# B&R Automation Studio project VisionSample (part 2)

#### brdkSTR.fun
```iecst
FUNCTION brdkStrAppendUdintToA : DINT (*Appends an UDINT to the end of a string. $RETURN=length;Length of the string.*) (*$GROUP=User,$CAT=User,$GROUPICON=User.png,$CATICON=User.png*)
	VAR_INPUT
		value : UDINT; (*UDINT value to be converted.*)
		pString : UDINT; (*String pointer to source string.*)
		base : USINT; (*0,10 = decimal, 2 = binary, 16 = hex.*)
		position : DINT; (*Append position. Negative numbers will count from end of string.*)
	END_VAR
END_FUNCTION

FUNCTION brdkStrAToDint : DINT (*Converts a string to a DINT type. $RETURN=value;DINT value.*) (*$GROUP=User,$CAT=User,$GROUPICON=User.png,$CATICON=User.png*)
	VAR_INPUT
		pString : UDINT; (*String pointer to source string.*)
		base : USINT; (*0,10 = decimal, 2 = binary, 16 = hex.*)
	END_VAR
END_FUNCTION

FUNCTION brdkStrAToUdint : UDINT (*Converts a string to an UDINT type. $RETURN=value;UDINT value.*) (*$GROUP=User,$CAT=User,$GROUPICON=User.png,$CATICON=User.png*)
	VAR_INPUT
		pString : UDINT; (*String pointer to source string.*)
		base : USINT; (*0,10 = decimal, 2 = binary, 16 = hex.*)
	END_VAR
END_FUNCTION

FUNCTION brdkStrCat : UDINT (*Appends a copy of the source string to the end of the destination string. $RETURN=address;Address after the string.*) (*$GROUP=User,$CAT=User,$GROUPICON=User.png,$CATICON=User.png*)
	VAR_INPUT
		pDestination : UDINT; (*Destination string pointer.*)
		pSource : UDINT; (*Source string pointer.*)
	END_VAR
END_FUNCTION

FUNCTION brdkStrCatAtChar : DINT (*Appends a copy of the source string to the char position of the destination string. $RETURN=index;Index in destination string where the source string is appended. -1 if char is not found.*) (*$GROUP=User,$CAT=User,$GROUPICON=User.png,$CATICON=User.png*)
	VAR_INPUT
		pDestination : UDINT; (*Destination string pointer.*)
		pSource : UDINT; (*Source string pointer.*)
		pChar : UDINT; (*Char pointer.*)
		direction : DINT; (*0 = first appearance of char, -1 = last appearance of char.*)
		greedy : BOOL; (*If true the source string is appended to the char position. If false the char is still present in the destination string.*)
	END_VAR
END_FUNCTION

FUNCTION brdkStrCharAt : USINT (*Returns the character at the specified index. $RETURN=coding;ASCII coding of the char.*) (*$GROUP=User,$CAT=User,$GROUPICON=User.png,$CATICON=User.png*)
	VAR_INPUT
		pString : UDINT; (*String pointer to source string.*)
		index : UDINT; (*Look up index.*)
		pChar : UDINT; (*Char pointer to char to look up.*)
	END_VAR
END_FUNCTION

FUNCTION brdkStrCharCount : DINT (*Finds how many times a character appears in a string. $RETURN=count;Char count. -1 if error.*) (*$GROUP=User,$CAT=User,$GROUPICON=User.png,$CATICON=User.png*)
	VAR_INPUT
		pString : UDINT; (*String pointer to source string.*)
		pChar : UDINT; (*Pointer to search char.*)
	END_VAR
END_FUNCTION

FUNCTION brdkStrCmp : DINT (*Compares character(s) from string1 to string2. $RETURN=result;0 means that the two string are equal.*)
	VAR_INPUT
		pString1 : UDINT; (*String1 pointer.*)
		pString2 : UDINT; (*String2 pointer.*)
	END_VAR
END_FUNCTION

FUNCTION brdkStrCpy : UDINT (*Copies a string to another string. $RETURN=address;Address after the string.*) (*$GROUP=User,$CAT=User,$GROUPICON=User.png,$CATICON=User.png*)
	VAR_INPUT
		pDestination : UDINT; (*Destination string pointer.*)
		pSource : UDINT; (*Source string pointer.*)
	END_VAR
END_FUNCTION

FUNCTION brdkStrCrc32 : UDINT (*Calculates a CRC32 checksum based on the input string. $RETURN=checksum;Checksum of the string.*) (*$GROUP=User,$CAT=User,$GROUPICON=User.png,$CATICON=User.png*)
	VAR_INPUT
		pString : UDINT; (*String pointer.*)
	END_VAR
END_FUNCTION

FUNCTION brdkStrDintToA : DINT (*Converts a DINT into a STRING type. $RETURN=length;Length of the string.*) (*$GROUP=User,$CAT=User,$GROUPICON=User.png,$CATICON=User.png*)
	VAR_INPUT
		value : DINT; (*DINT value to be converted.*)
		pString : UDINT; (*String pointer to source string.*)
		base : USINT; (*0,10 = decimal, 2 = binary, 16 = hex.*)
	END_VAR
END_FUNCTION

FUNCTION brdkStrEncode : DINT (*Encodes a string into different formats. $RETURN=address;Address after the string.*) (*$GROUP=User,$CAT=User,$GROUPICON=User.png,$CATICON=User.png*)
	VAR_INPUT
		pDestination : UDINT; (*Destination string pointer.*)
		pSource : UDINT; (*Source string pointer.*)
		format : USINT; (*0 = UTF-8*)
	END_VAR
END_FUNCTION

FUNCTION brdkStrFill : DINT (*Inserts amount of character(s) to the specified position of the string. $RETURN=length;Length of the string. -1 if error.*) (*$GROUP=User,$CAT=User,$GROUPICON=User.png,$CATICON=User.png*)
	VAR_INPUT
		pString : UDINT; (*String pointer to source string.*)
		amount : DINT; (*Fill char amount.*)
		pChar : UDINT; (*Fill char. If 0 whitespace is used.*)
		position : DINT; (*Fill position. Negative numbers will count from end of string.*)
	END_VAR
END_FUNCTION

FUNCTION brdkStrFillUp : DINT (*Fills x amount of character(s) to the specified position of the string. $RETURN=amount;Amount of chars filled. -1 if error.*) (*$GROUP=User,$CAT=User,$GROUPICON=User.png,$CATICON=User.png*)
	VAR_INPUT
		pString : UDINT; (*String pointer to source string.*)
		maxLength : DINT; (*Maximum length of the string.*)
		pChar : UDINT; (*Fill char. If 0 whitespace is used.*)
		position : DINT; (*Fill position. Negative numbers will count from end of string.*)
	END_VAR
END_FUNCTION

FUNCTION brdkStrIndexOf : DINT (*Returns the index within this string of the first or last occurrence of the specified character. $RETURN=index;Index of the char. -1 if char is not found.*) (*$GROUP=User,$CAT=User,$GROUPICON=User.png,$CATICON=User.png*)
	VAR_INPUT
		pString : UDINT; (*String pointer to source string.*)
		pChar : UDINT; (*Char pointer to char to look up.*)
		direction : DINT; (*0 = search from left, -1 = search from right.*)
	END_VAR
END_FUNCTION

FUNCTION brdkStrInsertAtPos : DINT (*Inserts a string into another string at a specified position. $RETURN=length;Length of the string. -1 if error.*) (*$GROUP=User,$CAT=User,$GROUPICON=User.png,$CATICON=User.png*)
	VAR_INPUT
		pString : UDINT; (*String pointer to source string.*)
		pInsert : UDINT; (*String pointer to insert string.*)
		position : DINT; (*Insert position. Negative numbers will count from end of string.*)
	END_VAR
END_FUNCTION

FUNCTION brdkStrIsAlphabet : BOOL (*Returns false or true depending of all characters are present in the alphabet. $RETURN=false/true; a..z = true.*) (*$GROUP=User,$CAT=User,$GROUPICON=User.png,$CATICON=User.png*)
	VAR_INPUT
		pString : UDINT; (*String pointer.*)
	END_VAR
END_FUNCTION

FUNCTION brdkStrIsDigit : BOOL (*Returns false or true depending of all characters are digits. $RETURN=false/true; 0..9 = true.*) (*$GROUP=User,$CAT=User,$GROUPICON=User.png,$CATICON=User.png*)
	VAR_INPUT
		pString : UDINT; (*String pointer.*)
	END_VAR
END_FUNCTION

FUNCTION brdkStrIsEmpty : BOOL (*Returns false or true depending of characters are present in the first position of the string. $RETURN=false/true;Position [0] = /0 = false. Position [0] != /0 = true.*) (*$GROUP=User,$CAT=User,$GROUPICON=User.png,$CATICON=User.png*)
	VAR_INPUT
		pString : UDINT; (*String pointer.*)
	END_VAR
END_FUNCTION

FUNCTION brdkStrJoin : DINT (*Joins elements from a string array into a string with a delimiter. $RETURN=length;Length of the string or error codes.*) (*$GROUP=User,$CAT=User,$GROUPICON=User.png,$CATICON=User.png*)
	VAR_INPUT
		pString : UDINT; (*String pointer to destination string.*)
		pArray : UDINT; (*Pointer to source string array.*)
		pDelimiter : UDINT; (*Delimiter char. If 0 whitespace is used. The delimiter can only be 1 char long.*)
		sizeOfArray : UDINT; (*Max. size of the string array. Size means number of elements in array.*)
		sizeOfArrayString : UDINT; (*Max. size of strings in the array.*)
		sizeOfString : UDINT; (*Max. size of destination string.*)
	END_VAR
END_FUNCTION

FUNCTION brdkStrLen : DINT (*Returns the number of characters in a string. Stops at \0. $RETURN=length;length of the string*) (*$GROUP=User,$CAT=User,$GROUPICON=User.png,$CATICON=User.png*)
	VAR_INPUT
		pString : UDINT; (*String pointer.*)
	END_VAR
END_FUNCTION

FUNCTION brdkStrMemClear : UDINT (*Fills amount of 0 to destination. $RETURN=address;Address after the destination.*) (*$GROUP=User,$CAT=User,$GROUPICON=User.png,$CATICON=User.png*)
	VAR_INPUT
		pDestination : UDINT; (*Destination pointer.*)
		amount : UDINT; (*Amount of character(s) to be initialized.*)
	END_VAR
END_FUNCTION

FUNCTION brdkStrMemCmp : DINT (*Compares amount of character(s) from area1 to area2. $RETURN=result;0 means that the two areas are equal.*) (*$GROUP=User,$CAT=User,$GROUPICON=User.png,$CATICON=User.png*)
	VAR_INPUT
		pArea1 : UDINT; (*Area1 pointer.*)
		pArea2 : UDINT; (*Area2 pointer.*)
		amount : UDINT; (*Amount of character(s) to be comared.*)
	END_VAR
END_FUNCTION

FUNCTION brdkStrMemCpy : UDINT (*Copies amount of character(s) from source to destination. $RETURN=address;Address after the destination.*) (*$GROUP=User,$CAT=User,$GROUPICON=User.png,$CATICON=User.png*)
	VAR_INPUT
		pDestination : UDINT; (*Destination pointer.*)
		pSource : UDINT; (*Source pointer.*)
		amount : UDINT; (*Amount of character(s) to be copied.*)
	END_VAR
END_FUNCTION

FUNCTION brdkStrMemMove : UDINT (*Moves amount of character(s) from source to destination. $RETURN=address;Address after the destination.*) (*$GROUP=User,$CAT=User,$GROUPICON=User.png,$CATICON=User.png*)
	VAR_INPUT
		pDestination : UDINT; (*Destination pointer.*)
		pSource : UDINT; (*Source pointer.*)
		amount : UDINT; (*Amount of character(s) to be moved.*)
	END_VAR
END_FUNCTION

FUNCTION brdkStrMemSet : UDINT (*Fills amount of character(s) to destination. $RETURN=address;Address after the destination.*) (*$GROUP=User,$CAT=User,$GROUPICON=User.png,$CATICON=User.png*)
	VAR_INPUT
		pDestination : UDINT; (*Destination pointer.*)
		value : USINT; (*Initialization value.*)
		amount : UDINT; (*Amount of character(s) to be initialized.*)
	END_VAR
END_FUNCTION

FUNCTION brdkStrMove : UDINT (*Moves a string to another string. $RETURN=address;Address after the string.*) (*$GROUP=User,$CAT=User,$GROUPICON=User.png,$CATICON=User.png*)
	VAR_INPUT
		pDestination : UDINT; (*Destination string pointer.*)
		pSource : UDINT; (*Source string pointer.*)
	END_VAR
END_FUNCTION

FUNCTION brdkStrNCpy : UDINT (*Copies a string to another string. If the function encounters a null character in the source string, the function will add null characters to the destination string until amount character(s) have been written. $RETURN=address;Address after the string.*) (*$GROUP=User,$CAT=User,$GROUPICON=User.png,$CATICON=User.png*)
	VAR_INPUT
		pDestination : UDINT; (*Destination string pointer.*)
		pSource : UDINT; (*Source string pointer.*)
		amount : UDINT; (*Amount of character(s) to be moved.*)
	END_VAR
END_FUNCTION

FUNCTION brdkStrRemove : UDINT (*Removes character(s) from a string from a specified position. $RETURN=address;Address after the string.*) (*$GROUP=User,$CAT=User,$GROUPICON=User.png,$CATICON=User.png*)
	VAR_INPUT
		pString : UDINT; (*Source string pointer.*)
		start : DINT; (*Index of where to start in the string. Negative numbers start from the end of the string.*)
		length : DINT; (*0 means to the end of the string. Negative length is subtracted from the end of the string. Is start is negative length is subtracted from the start of the string. *)
	END_VAR
END_FUNCTION

FUNCTION brdkStrRepeat : DINT (*Repeats a string a specified number of times. $RETURN=length;Length of the string.*) (*$GROUP=User,$CAT=User,$GROUPICON=User.png,$CATICON=User.png*)
	VAR_INPUT
		pString : UDINT; (*String pointer to source string.*)
		times : DINT; (*Number of times the string should be repeated.*)
	END_VAR
END_FUNCTION

FUNCTION brdkStrReplace : DINT (*Replaces some characters with some other characters in a string. $RETURN=number;Number of replacements done.*) (*$GROUP=User,$CAT=User,$GROUPICON=User.png,$CATICON=User.png*)
	VAR_INPUT
		pString : UDINT; (*String pointer to source string.*)
		pFind : UDINT; (*String pointer to find string.*)
		pReplace : UDINT; (*String pointer to replacement string:*)
	END_VAR
END_FUNCTION

FUNCTION brdkStrReverse : DINT (*Reverses a string from start position to end position. $RETURN=count;Number of reverses done. -1 if error.*) (*$GROUP=User,$CAT=User,$GROUPICON=User.png,$CATICON=User.png*)
	VAR_INPUT
		pString : UDINT; (*String pointer to source string.*)
		startPosition : DINT; (*Start position. Must be a positive number and less than length.*)
		endPosition : DINT; (*End position. Must be less than length unless it's a negative numbers which will count from end of string.*)
	END_VAR
END_FUNCTION

FUNCTION brdkStrReverseWords : DINT (*Reverses words in a string. $RETURN=count;Number of words reversed.*) (*$GROUP=User,$CAT=User,$GROUPICON=User.png,$CATICON=User.png*)
	VAR_INPUT
		pString : UDINT; (*String pointer to source string.*)
	END_VAR
END_FUNCTION

FUNCTION brdkStrSearch : DINT (*Searches a string for a specified string. $RETURN=position; Position of the match. -1 if no match.*) (*$GROUP=User,$CAT=User,$GROUPICON=User.png,$CATICON=User.png*)
	VAR_INPUT
		pString : UDINT; (*String pointer to source string.*)
		pSearchString : UDINT; (*String pointer to search string.*)
	END_VAR
END_FUNCTION

FUNCTION brdkStrSlice : DINT (*Slices a part of a string. $RETURN=length;Length of the string. -1 if error.*) (*$GROUP=User,$CAT=User,$GROUPICON=User.png,$CATICON=User.png*)
	VAR_INPUT
		pString : UDINT; (*String pointer to source string.*)
		start : DINT; (*Start position.*)
		end : DINT; (*End position.*)
	END_VAR
END_FUNCTION

FUNCTION brdkStrSplit : DINT (*Splits a string into an array of string using a seperator. $RETURN=count;Number of elements splitted or an error code.*) (*$GROUP=User,$CAT=User,$GROUPICON=User.png,$CATICON=User.png*)
	VAR_INPUT
		pArray : UDINT; (*Pointer to destination string array.*)
		pString : UDINT; (*String pointer to source string.*)
		pDelimiter : UDINT; (*Delimiter char. If 0 whitespace is used. The delimiter can only be 1 char long.*)
		sizeOfArray : UDINT; (*Max. size of the string array. Size means number of elements in array.*)
		sizeofArrayString : UDINT; (*Max. size of strings in the array.*)
		greedy : BOOL; (*Remove or keep the seperator from the string.*)
	END_VAR
END_FUNCTION

FUNCTION brdkStrSubDintSearch : DINT (*Returns a DINT based on a search. $RETURN=length;Length of the destination string. -1 if error.*) (*$GROUP=User,$CAT=User,$GROUPICON=User.png,$CATICON=User.png*)
	VAR_INPUT
		pSource : UDINT; (*Source string pointer.*)
		pStart : UDINT; (*String pointer for start search string.*)
		pEnd : UDINT; (*String pointer for end search string. The function will only search after the start string.*)
		startOffset : DINT; (*Offset for the start poition. If greedy = true offset is after the start has been removed.*)
		base : USINT; (*0,10 = decimal, 2 = binary, 16 = hex.*)
	END_VAR
END_FUNCTION

FUNCTION brdkStrSubStr : DINT (*Returns a part of a string. $RETURN=length;Length of the destination string. -1 if error.*) (*$GROUP=User,$CAT=User,$GROUPICON=User.png,$CATICON=User.png*)
	VAR_INPUT
		pDestination : UDINT; (*Destination string pointer.*)
		pSource : UDINT; (*Source string pointer.*)
		start : DINT; (*Index of where to start in the string. Negative numbers start from the end of the string.*)
		length : DINT; (*0 means to the end of the string. Negative length is subtracted from the end of the string. Is start is negative length is subtracted from the start of the string. *)
	END_VAR
END_FUNCTION

FUNCTION brdkStrSubStrSearch : BOOL (*Returns a part of a string based on a search. $RETURN=success;TRUE = success *) (*$GROUP=User,$CAT=User,$GROUPICON=User.png,$CATICON=User.png*)
	VAR_INPUT
		pDestination : UDINT; (*Destination string pointer.*)
		pSource : UDINT; (*Source string pointer.*)
		pStart : UDINT; (*String pointer for start search string.*)
		pEnd : UDINT; (*String pointer for end search string. The function will only search after the start string.*)
		startOffset : DINT; (*Offset for the start poition. If greedy = true offset is after the start has been removed.*)
		greedy : BOOL; (*Will add or remove the search strings from the destination string.*)
	END_VAR
END_FUNCTION

FUNCTION brdkStrToDec : DINT (*Converts a string of hexadecimal values to ASCII characters. $RETURN=length;Length of the string. -1 if error.*) (*$GROUP=User,$CAT=User,$GROUPICON=User.png,$CATICON=User.png*)
	VAR_INPUT
		pString : UDINT; (*String pointer to source string.*)
	END_VAR
END_FUNCTION

FUNCTION brdkStrToHex : DINT (*Converts a string of ASCII characters to hexadecimal values. $RETURN=length;Length of the string.*) (*$GROUP=User,$CAT=User,$GROUPICON=User.png,$CATICON=User.png*)
	VAR_INPUT
		pString : UDINT; (*String pointer to source string.*)
	END_VAR
END_FUNCTION

FUNCTION brdkStrToLowerCase : DINT (*Converts a string to lowercase letters. $RETURN=number;Number of characters changed.*) (*$GROUP=User,$CAT=User,$GROUPICON=User.png,$CATICON=User.png*)
	VAR_INPUT
		pString : UDINT; (*String pointer to source string.*)
	END_VAR
END_FUNCTION

FUNCTION brdkStrToUpperCase : DINT (*Converts a string to uppercase letters. $RETURN=number;Number of characters changed.*) (*$GROUP=User,$CAT=User,$GROUPICON=User.png,$CATICON=User.png*)
	VAR_INPUT
		pString : UDINT; (*String pointer to source string.*)
	END_VAR
END_FUNCTION

FUNCTION brdkStrToUpperCaseWords : DINT (*Convert the first character of each word to uppercase. (title()). $RETURN=number;Number of characters changed.*) (*$GROUP=User,$CAT=User,$GROUPICON=User.png,$CATICON=User.png*)
	VAR_INPUT
		pString : UDINT; (*String pointer to source string.*)
	END_VAR
END_FUNCTION

FUNCTION brdkStrTrim : DINT (*Removes whitespaces from a string. $RETURN=number;Number of whitespaces removed from string.*) (*$GROUP=User,$CAT=User,$GROUPICON=User.png,$CATICON=User.png*)
	VAR_INPUT
		pString : UDINT; (*String pointer to source string.*)
		direction : DINT; (*0 = both sides, 1 = left side only, -1 = right side only.*)
	END_VAR
END_FUNCTION

FUNCTION brdkStrUdintToA : DINT (*Converts an UDINT into a STRING type. $RETURN=length;Length of the string.*) (*$GROUP=User,$CAT=User,$GROUPICON=User.png,$CATICON=User.png*)
	VAR_INPUT
		value : UDINT; (*UDINT value to be converted.*)
		pString : UDINT; (*String pointer to source string.*)
		base : USINT; (*0,10 = decimal, 2 = binary, 16 = hex.*)
	END_VAR
END_FUNCTION

FUNCTION brdkStrWord : DINT (*Returns a word in a string given by a number and a delimiter. $RETURN=length;Length of the string.*) (*$GROUP=User,$CAT=User,$GROUPICON=User.png,$CATICON=User.png*)
	VAR_INPUT
		pDestination : UDINT; (*Destination string pointer.*)
		pSource : UDINT; (*Source string pointer.*)
		pDelimiter : UDINT; (*Delimiter char. If 0 whitespace is used. The delimiter can only be 1 char long.*)
		number : DINT; (*Word number in string. 1 = first word. -1 = last word.*)
		sizeOfString : UDINT; (*Max. size of destination string.*)
	END_VAR
END_FUNCTION
```

#### brdkStrAppendUdintToA.c
```c
#include <brdkSTR_func.h>

signed long brdkStrAppendUdintToA(unsigned long value, unsigned long pString, unsigned char base, signed long position) {
	signed long i,cnt=0,len = brdkStrLen(pString);
	signed long start = position > -1 ? position :len+position+1;
	unsigned char tmp;
	i=start;
	tmp = 0x30;
	base = !base ? 10 : base;	/* make sure base is not 0 */
	if (value != 0) {
		while (value > 0) {
			unsigned long rem = value % base;
			unsigned char tmp = (rem > 9)? (rem-10) + 0x41 : rem + 0x30;	/* 0x41 = A, 0x30 = 0*/
			brdkStrFill(pString,1,(unsigned long)&tmp,i++);
	       	value = value/base;
			cnt++;
		}
		brdkStrReverse(pString,start,--i);
		return len+cnt;
	}
	else {
		brdkStrFill(pString,1,(unsigned long)&tmp,i);
		return len+1;
	}
}
```

#### brdkStrAToDint.c
```c
#include <brdkSTR_func.h>

signed long brdkStrAToDint(unsigned long pString, unsigned char base) {
	/* check if string starts with a minus sign */
	if(((char*)pString)[0] == 0x2d) return -brdkStrAToUdint(pString+1,BRDK_STR_CONVERT_DECIMAL);
	else return brdkStrAToUdint(pString,base);
}
```

#### brdkStrAToUdint.c
```c
#include <brdkSTR_func.h>

unsigned long brdkStrAToUdint(unsigned long pString, unsigned char base) {
	signed long len = brdkStrLen(pString);
	return aToUdint(pString, len, base);
}
```

#### brdkStrCat.c
```c
#include <brdkSTR_func.h>

unsigned long brdkStrCat(unsigned long pDestination, unsigned long pSource) {
	unsigned long i=0,len = brdkStrLen(pSource), start = brdkStrLen(pDestination);
	for(i=0; i< len; i++) ((char*)pDestination)[start+i] = ((char*)pSource)[i];
	((char*)pDestination)[start+i] = 0;
	return pDestination+start+i;
}
```

#### brdkStrCatAtChar.c
```c
#include <brdkSTR_func.h>

signed long brdkStrCatAtChar(unsigned long pDestination, unsigned long pSource, unsigned long pChar, signed long direction, unsigned char greedy) {
	unsigned long i=0,len = brdkStrLen(pSource);
	signed long start = brdkStrIndexOf(pDestination,pChar,direction);
	if(start > -1) {
		start += !greedy;
		for(i=0; i< len; i++) ((char*)pDestination)[start+i] = ((char*)pSource)[i];
		((char*)pDestination)[start+i] = 0;
	}
	return start;
}
```

#### brdkStrCharAt.c
```c
#include <brdkSTR_func.h>

unsigned char brdkStrCharAt(unsigned long pString, unsigned long index, unsigned long pChar) {
	if(index < brdkStrLen(pString)) {
		*(char*)pChar = ((char*)pString)[index];
		return ((char*)pString)[index];
	}
	else {
		*(char*)pChar = 0;
		return 0;
	}
}
```

#### brdkStrCharCount.c
```c
#include <brdkSTR_func.h>

signed long brdkStrCharCount(unsigned long pString, unsigned long pChar) {
	signed long i=0, cnt=0;
	if(pChar != 0 && *(char*)pChar != 0) {
		while(((char*)pString)[i]) if(((char*)pString)[i++] == *(char*)pChar) cnt++;
	}
	else cnt = -1;
	return cnt;
}
```

#### brdkStrCmp.c
```c
#include <brdkSTR_func.h>

signed long brdkStrCmp(unsigned long pString1, unsigned long pString2) {
	unsigned long i=0;
	do if(((char*)pString1)[i] != ((char*)pString2)[i]) break;
	while(((char*)pString1)[i] != 0 && ((char*)pString2)[i++] != 0);
	return ((char*)pString1)[i]-((char*)pString2)[i];
}
```

#### brdkStrCpy.c
```c
#include <brdkSTR_func.h>

unsigned long brdkStrCpy(unsigned long pDestination, unsigned long pSource) {
	unsigned long i=0;
	do ((char*)pDestination)[i] = ((char*)pSource)[i];
	while(((char*)pSource)[i++] != 0);
	return pDestination+i;
}
```

#### brdkStrCrc32.c
```c
#include <brdkSTR_func.h>

unsigned long brdkStrCrc32(unsigned long pString) {
	int i=0, crc = 0xFFFFFFFF;
	unsigned int byte, c;
	const unsigned int g0 = 0xEDB88320, g1 = g0>>1,g2 = g0>>2, g3 = g0>>3, g4 = g0>>4, g5 = g0>>5, g6 = (g0>>6)^g0, g7 = ((g0>>6)^g0)>>1;
	while ((byte = ((char*)pString)[i]) != 0) {    /* Get next byte. */
		crc = crc ^ byte;
		c = ((crc<<31>>31) & g7) ^ ((crc<<30>>31) & g6) ^
			((crc<<29>>31) & g5) ^ ((crc<<28>>31) & g4) ^
			((crc<<27>>31) & g3) ^ ((crc<<26>>31) & g2) ^
			((crc<<25>>31) & g1) ^ ((crc<<24>>31) & g0);
		crc = ((unsigned)crc >> 8) ^ c;
		i++;
   }
   return ~crc;
}
```

#### brdkStrDintToA.c
```c
#include <brdkSTR_func.h>

signed long brdkStrDintToA(signed long value, unsigned long pString, unsigned char base) {
	if(value < 0) {
		((char*)pString)[0] = 0x2d; /* - sign */
		return brdkStrUdintToA(-value,pString+1,BRDK_STR_CONVERT_DECIMAL)+1;
	}
	else return brdkStrUdintToA(value,pString,base);
}
```

#### brdkStrEncode.c
```c
#include <brdkSTR_func.h>

signed long brdkStrEncode(unsigned long pDestination, unsigned long pSource, unsigned char format) {
	unsigned long i=0;
	switch(format) {
		case BRDK_STR_UTF_8:

			do ((unsigned char*)pDestination)[i] = ((unsigned char*)pSource)[i] <= 127 ? ((unsigned char*)pSource)[i] : ((unsigned char*)pSource)[i] + 35;
			while(((char*)pSource)[i++] != 0);
			return pDestination+i;
			break;

		default:
			return -1;
			break;
	}
}
```

#### brdkStrFill.c
```c
#include <brdkSTR_func.h>

signed long brdkStrFill(unsigned long pString, signed long amount, unsigned long pChar, signed long position) {
	signed long i,j, len = brdkStrLen(pString), tmpPos;
	char ch;
	i = len+amount;
	j = len;
	ch = pChar != 0 && *(char*)pChar != 0 ? *(char*)pChar : 0x20;	/* white space is default */
	tmpPos = position >= 0 ? position : len + 1 + position;
	if(tmpPos > -1) {
		while(j>=tmpPos) ((char*)pString)[i--] = ((char*)pString)[j--];
		while(i>=tmpPos) ((char*)pString)[i--] = ch;
		return len+amount;
	}
	else return -1;
}
```

#### brdkStrFillUp.c
```c
#include <brdkSTR_func.h>

signed long brdkStrFillUp(unsigned long pString, signed long maxLength, unsigned long pChar, signed long position) {
	signed long amount = maxLength-brdkStrLen(pString);
	if(amount > 0) {
		if(brdkStrFill(pString, amount, pChar, position) != -1) return amount;
		else return -1;
	}
	return 0;
}
```

#### brdkStrIndexOf.c
```c
#include <brdkSTR_func.h>

signed long brdkStrIndexOf(unsigned long pString, unsigned long pChar, signed long direction) {
	signed long i;
	if(direction > -1) {
		i = 0;
		while(((char*)pString)[i]) {
			if(((char*)pString)[i] == ((char*)pChar)[0]) break;
			else i++;
		}
		if(((char*)pString)[i] != 0) return i;
		else return -1;
	}
	else {
		i = brdkStrLen(pString)-1;
		while(((char*)pString)[i] && i > -1) if(((char*)pString)[i--] == ((char*)pChar)[0]) break;
		if(((char*)pString)[i] != 0) return ++i;
		else return -1;
	}
}
```

#### brdkStrInsertAtPos.c
```c
#include <brdkSTR_func.h>

signed long brdkStrInsertAtPos(unsigned long pString, unsigned long pInsert, signed long position) {
	signed long i,j, len = brdkStrLen(pString), lenIns = brdkStrLen(pInsert), tmpPos;
	if(lenIns > 0) {
		if(len==0 && (position==0 || position==-1)){
			i=0;
			while(((char*)pInsert)[i]) {
				((char*)pString)[i] = ((char*)pInsert)[i];
				i++;
			}
			((char*)pString)[i] = 0;
			len = i;
		}
		else if(position <= len) {
			i = len+lenIns;
			j = len;
			tmpPos = position >= 0 ? position : len + 1 + position;
			if(tmpPos > -1) {
				while(j>=tmpPos) ((char*)pString)[i--] = ((char*)pString)[j--];
				j=lenIns-1;
				while(i>=tmpPos) ((char*)pString)[i--] = ((char*)pInsert)[j--];
				len+=lenIns;
			}
			else len = -1;
		}
	}
	return len;
}
```

#### brdkStrIsAlphabet.c
```c
#include <brdkSTR_func.h>

unsigned char brdkStrIsAlphabet(unsigned long pString) {
	unsigned long len = 0;
	while(((char*)pString)[len]) {
		if (((char*)pString)[len] > 0x5A) {	/* is it larger that Z */
			if(((char*)pString)[len] < 0x61 || 0x7a < ((char*)pString)[len]) return 0;
		}
		else if(((char*)pString)[len] < 0x41) return 0;		/* is it smaller than A */
		len++;
	}
	return 1;
}
```

#### brdkStrIsDigit.c
```c
#include <brdkSTR_func.h>

unsigned char brdkStrIsDigit(unsigned long pString) {
	unsigned long len = 0;
	while(((char*)pString)[len]) {
		if (((char*)pString)[len] < 0x30 || 0x39 < ((char*)pString)[len]) return 0;
		len++;
	}
	return 1;
}
```

#### brdkStrIsEmpty.c
```c
#include <brdkSTR_func.h>

unsigned char brdkStrIsEmpty(unsigned long pString) {
	return ((char*)pString)[0] == 0;
}
```

#### brdkStrJoin.c
```c
#include <brdkSTR_func.h>

signed long brdkStrJoin(unsigned long pString, unsigned long pArray, unsigned long pDelimiter, unsigned long sizeOfArray, unsigned long sizeOfArrayString, unsigned long sizeOfString) {
	unsigned long sIdx = 0, pArr = pArray, aIdx = 0;
	if(pArray != 0 && pString != 0 && sizeOfArray != 0 && sizeOfArrayString != 0) {		/* check all pointers are set */
		if(pDelimiter == 0) pDelimiter = (unsigned long)" ";							/* use white space is delimiter pointer is 0 */
		while(((char*)pArr)[0] != 0) {													/* continue until we find the first empty array string */
			if(((char*)pArr)[aIdx] != 0) {
				((char*)pString)[sIdx++] = ((char*)pArr)[aIdx++];						/* copy string data */
				if(sIdx >= sizeOfString) return -2;										/* destination string too small */
			}
			else {
				pArr += sizeOfArrayString;												/* jump to the next array element */
				aIdx = 0;
				((char*)pString)[sIdx++] = ((char*)pDelimiter)[0];						/* insert delimiter */
				if(sIdx >= sizeOfString) return -2;										/* destination string too small */
				if(pArr > (pArray + sizeOfArray)) {										/* we hit the end of the array */
					break;
				}
			}
		}
		if(sIdx == 0) return 0;															/* nothing copied */
		sIdx--;
		((char*)pString)[sIdx] = 0;														/* end the string. -e because we inserted a delimiter at the end */
		return sIdx;
	}
	else return -1;
	return -4;
}
```

#### brdkStrLen.c
```c
#include <brdkSTR_func.h>

signed long brdkStrLen(unsigned long pString) {
	unsigned long len = 0;
	while(((char*)pString)[len]) len++;	/* makes a little strlen */
	return len;
}
```

#### brdkStrMemClear.c
```c
#include <brdkSTR_func.h>

unsigned long brdkStrMemClear(unsigned long pDestination, unsigned long amount) {
	return brdkStrMemSet(pDestination,0,amount);
}
```

#### brdkStrMemCmp.c
```c
#include <brdkSTR_func.h>

signed long brdkStrMemCmp(unsigned long pString1, unsigned long pString2, unsigned long amount) {
	unsigned long i=0;
	for(i=0; i< amount; i++) if(((char*)pString1)[i] != ((char*)pString2)[i]) break;
	return ((char*)pString1)[i]-((char*)pString2)[i];
}
```

#### brdkStrMemCpy.c
```c
#include <brdkSTR_func.h>

unsigned long brdkStrMemCpy(unsigned long pDestination, unsigned long pSource, unsigned long amount) {
	unsigned long i=0;
	for(i=0; i< amount; i++) ((char*)pDestination)[i] = ((char*)pSource)[i];
	return pDestination+amount;
}
```

#### brdkStrMemMove.c
```c
#include <brdkSTR_func.h>

unsigned long brdkStrMemMove(unsigned long pDestination, unsigned long pSource, unsigned long amount) {
	unsigned long i=0;
	char buffer[amount];	/* if the destination and source is the same string we need a buffer */
	for(i=0; i< amount; i++) buffer[i] = ((char*)pSource)[i];
	for(i=0; i< amount; i++) ((char*)pDestination)[i] = buffer[i];
	return pDestination+amount;
}
```

#### brdkStrMemSet.c
```c
#include <brdkSTR_func.h>

unsigned long brdkStrMemSet(unsigned long pDestination, unsigned char value, unsigned long amount) {
	unsigned long i=0;
	for(i=0; i< amount; i++) ((char*)pDestination)[i] = value;
	return pDestination+amount;
}
```

#### brdkStrMove.c
```c
#include <brdkSTR_func.h>

unsigned long brdkStrMove(unsigned long pDestination, unsigned long pSource) {
	return brdkStrMemMove(pDestination,pSource,brdkStrLen(pSource));
}
```

#### brdkStrNCpy.c
```c
#include <brdkSTR_func.h>

unsigned long brdkStrNCpy(unsigned long pDestination, unsigned long pSource, unsigned long amount) {
	unsigned long i=0;
	for(i=0; i< amount; i++) {
		if(((char*)pSource)[i]) ((char*)pDestination)[i] = ((char*)pSource)[i];
		else ((char*)pDestination)[i] = 0;
	}
	return pDestination+amount;
}
```

#### brdkStrRemove.c
```c
#include <brdkSTR_func.h>

unsigned long brdkStrRemove(unsigned long pString, signed long start, signed long length) {
	signed long end, len=0;
	if(start < 0) {
		len = brdkStrLen(pString);
		if(length<1) {
			len = start;
			start = length*(-1);
			length = brdkStrLen(pString)-start+len+1;
		}
		else start = len+start-length+1;
	}
	else if(length<1) length = brdkStrLen(pString)-start+length;
	end = start+length;
	while(((char*)pString)[end]) ((char*)pString)[start++] = ((char*)pString)[end++];
	((char*)pString)[start] = 0;
	return pString+start+1;
}
```

#### brdkStrRepeat.c
```c
#include <brdkSTR_func.h>

signed long brdkStrRepeat(unsigned long pString, signed long times) {
	signed long i,j,t,len = brdkStrLen(pString);
	j=len;
	for(t=0; t < times; t++) {
		for(i=0; i< len; i++) ((char*)pString)[j+i] = ((char*)pString)[i];
		j += len;
	}
	((char*)pString)[j] = 0;
	return j;
}
```

#### brdkStrReplace.c
```c
#include <brdkSTR_func.h>

signed long brdkStrReplace(unsigned long pString, unsigned long pFind, unsigned long pReplace) {
	signed long i=0, cnt=0, lenF = brdkStrLen(pFind), lenR = brdkStrLen(pReplace);
	i = brdkStrSearch(pString,pFind);
	while(i > -1) {
		brdkStrRemove(pString,i,lenF);
		brdkStrInsertAtPos(pString,pReplace,i);
		pString += i + lenR;
		i = brdkStrSearch(pString,pFind);
		cnt++;
	}
	return cnt;
}
```

#### brdkStrReverse.c
```c
#include <brdkSTR_func.h>

signed long brdkStrReverse(unsigned long pString, signed long startPosition, signed long endPosition) {
	signed long start = -1, end = -1, len = brdkStrLen(pString), cnt = 0;
    unsigned char tmp;
	/* make sure start position is valid */
	if(startPosition > -1 && startPosition < len) start = startPosition;
	else return -1;
	/* make sure end position is valid */
	if(endPosition > -1 && endPosition < len && endPosition > startPosition) end = endPosition;
	else if(endPosition < 0) end = len + endPosition;
	else return -1;
	while (start < end) {
        tmp = ((char*)pString)[start];
        ((char*)pString)[start++] = ((char*)pString)[end];
        ((char*)pString)[end--] = tmp;
		cnt++;
    }
	return cnt;
}
```

#### brdkStrReverseWords.c
```c
#include <brdkSTR_func.h>

signed long brdkStrReverseWords(unsigned long pString) {
	signed long i=0,wordPos=-1, cnt=0;
	while(((char*)pString)[i]) {
		if(wordPos<0 && (((char*)pString)[i] != 0x20)) wordPos = i;
		if(wordPos>-1 && (((char*)pString)[i+1] == 0x20 || ((char*)pString)[i+1] == 0)) {
			brdkStrReverse(pString,wordPos,i);
            wordPos = -1;
			cnt++;
        }
		i++;
	}
	brdkStrReverse(pString,0,i-1);
	return cnt;
}
```

#### brdkStrSearch.c
```c
#include <brdkSTR_func.h>

signed long brdkStrSearch(unsigned long pString, unsigned long pSearchString) {
	signed long lenString = brdkStrLen(pString), lenSearch = brdkStrLen(pSearchString);
	return search(pString, lenString, pSearchString, lenSearch);
}
```

#### brdkStrSlice.c
```c
#include <brdkSTR_func.h>

signed long brdkStrSlice(unsigned long pString, signed long start, signed long end) {
	signed long i,j, len = -1;
	if(start > -1) {
		if(start > 0) {
			len = brdkStrLen(pString);
			j=0;
			while(j<start) {
				for(i=0;i < len;i++) ((char*)pString)[i] = ((char*)pString)[i+1];	/* moves all characters one place left */
				len--;
				j++;
			}
		}
		if(end > 0) {
			end -= start;
			((char*)pString)[end] = 0;
			len = end;
		}
		else if(end < 0) {
			len = brdkStrLen(pString);
			if((end*(-1))<=len) {
				len += end;
				((char*)pString)[len+1+end] = 0;
			}
		}
		return len;
	}
	else return -1;
}
```

#### brdkStrSplit.c
```c
#include <brdkSTR_func.h>

signed long brdkStrSplit(unsigned long pArray, unsigned long pString, unsigned long pDelimiter, unsigned long sizeOfArray, unsigned long sizeOfArrayString, unsigned char greedy) {
	signed long size = 0;
	if(pArray != 0 && pString != 0 && sizeOfArray != 0 && sizeOfArrayString != 0) {		/* check all pointers are set */
		if(pDelimiter == 0) pDelimiter = (unsigned long)" ";							/* use white space is delimiter pointer is 0 */
		unsigned long i = 0, pArr = pArray, aIdx = 0;
		while(((char*)pString)[i] != 0) {												/* run while we dopn't hit a 0 */
			if(((char*)pString)[i] != ((char*)pDelimiter)[0]) {							/* check for delimiter */
				((char*)pArr)[aIdx++] = ((char*)pString)[i++];
				if(aIdx >= sizeOfArrayString) return -2;								/* array string too small */
			}
			else {
				if(!greedy) ((char*)pArr)[aIdx++] = ((char*)pString)[i];				/* check is delimiter should be removed */
				i++;
				if(aIdx >= sizeOfArrayString) return -2;								/* array string too small */
				((char*)pArr)[aIdx] = 0;
				pArr += sizeOfArrayString;												/* jump to the next array element */
				aIdx = 0;
				size++;
				if(pArr > (pArray + sizeOfArray)) return -3;							/* array too small */
			}
		}
		((char*)pArr)[aIdx] = 0;
		pArr += sizeOfArrayString;														/* jump to the next array element */
		size++;
		while(pArr < (pArray + sizeOfArray)) {											/* set the rest of the array elements to '' */
			((char*)pArr)[0] = 0;
			pArr += sizeOfArrayString;
		}
		return size;
	}
	else return -1;
	return -4;
}
```

#### brdkStrSubDintSearch.c
```c
#include <brdkSTR_func.h>

signed long brdkStrSubDintSearch(unsigned long pSource, unsigned long pStart, unsigned long pEnd, signed long startOffset, unsigned char base) {
	signed long posEnd, lenSource = brdkStrLen(pSource), lenStart = brdkStrLen(pStart), lenEnd, posGreedyStartOffset;
	signed long posStart = search(pSource, lenSource, pStart, lenStart);
	if(posStart > -1) {
		lenEnd = brdkStrLen(pEnd);
		posGreedyStartOffset = posStart + lenStart + startOffset;
		posEnd = search((unsigned long)&((char*)pSource)[posGreedyStartOffset], lenSource-posGreedyStartOffset, pEnd, lenEnd);
		if(posEnd > -1) {
			/* check if string starts with a minus sign */
			if(((char*)pSource)[posGreedyStartOffset] == 0x2d) return -aToUdint((unsigned long)&((char*)pSource)[posGreedyStartOffset+1],posEnd,base);
			else return aToUdint((unsigned long)&((char*)pSource)[posGreedyStartOffset],posEnd,base);
		}
	}
	return -1;
}
```

#### brdkStrSubStr.c
```c
#include <brdkSTR_func.h>

signed long brdkStrSubStr(unsigned long pDestination, unsigned long pSource, signed long start, signed long length) {
	signed long i=0,len=0;
	char buffer[length];	/* if the destination and source is the same string we need a buffer */
	if(start < 0) {
		len = brdkStrLen(pSource);
		if(length<1) {
			len = start;
			start = length*(-1);
			length = brdkStrLen(pSource)-start+len+1;
		}
		else start = len+start-length+1;
	}
	else if(length<1) length = brdkStrLen(pSource)-start+length;
	for(i=0; i< length; i++) buffer[i] = ((char*)pSource)[start+i];
	for(i=0; i< length; i++) ((char*)pDestination)[i] = buffer[i];
	((char*)pDestination)[i] = 0;
	return length;
}
```

#### brdkStrSubStrSearch.c
```c
#include <brdkSTR_func.h>

unsigned char brdkStrSubStrSearch(unsigned long pDestination, unsigned long pSource, unsigned long pStart, unsigned long pEnd, signed long startOffset, unsigned char greedy) {
	signed long posEnd, lenSource = brdkStrLen(pSource), lenStart = brdkStrLen(pStart), lenEnd, posGreedyStartOffset;
	signed long posStart = search(pSource, lenSource, pStart, lenStart);
	if(posStart > -1) {
		lenEnd = brdkStrLen(pEnd);
		posGreedyStartOffset = posStart + lenStart + startOffset;
		posEnd = search((unsigned long)&((char*)pSource)[posGreedyStartOffset], lenSource-posGreedyStartOffset, pEnd, lenEnd);
		if(posEnd > -1) {
			if(!greedy) {
				posGreedyStartOffset = posStart;
				posEnd += lenStart + startOffset + 1;
			}
			brdkStrMemCpy(pDestination, (unsigned long)&((char*)pSource)[posGreedyStartOffset],posEnd);
			((char*)pDestination)[posEnd] = 0;
			return 1;
		}
	}
	return 0;
}
```

#### brdkStrToDec.c
```c
#include <brdkSTR_func.h>

signed long brdkStrToDec(unsigned long pString) {
	signed long i=0,j=0;
	while(((char*)pString)[i]) {
		if(((char*)pString)[i+1] != 0) {
			char tmp[3];
			tmp[0] = ((char*)pString)[i++];
			tmp[1] = ((char*)pString)[i++];
			tmp[2] = 0;
			((char*)pString)[j++] = brdkStrAToUdint((unsigned long)&tmp, BRDK_STR_CONVERT_HEX);
		}
		else {
			i = -1;
			break;
		}
		((char*)pString)[j] = 0;
	}
	return i;
}
```

#### brdkStrToHex.c
```c
#include <brdkSTR_func.h>

signed long brdkStrToHex(unsigned long pString) {
	signed long i=0;
	unsigned long rem;
	unsigned char tmp;
	while(((char*)pString)[i]) {
		unsigned char value = (unsigned char)((char*)pString)[i];
		if(value < 0x10) {															/* a character with value below 9 we want representated with a 0 in front */
			brdkStrFill(pString,1,(unsigned long)&"0",i++);
			rem = value % 16;
		    ((char*)pString)[i++] = (rem > 9)? (rem-10) + 0x41 : rem + 0x30;		/* 0x41 = A, 0x30 = 0*/
		}
		else {
			while(value > 0) {
				rem = value % 16;
		       	((char*)pString)[i++] = (rem > 9)? (rem-10) + 0x41 : rem + 0x30;	/* 0x41 = A, 0x30 = 0*/
		       	value = value/16;
				if(value > 0) brdkStrFill(pString,1,(unsigned long)&" ",i);
				else {
					/* swap places */
					tmp = ((char*)pString)[i-1];
					((char*)pString)[i-1] = ((char*)pString)[i-2];
					((char*)pString)[i-2] = tmp;
				}
			}
		}
	}
	((char*)pString)[i] = 0;
	return i;
}
```

#### brdkStrToLowerCase.c
```c
#include <brdkSTR_func.h>

signed long brdkStrToLowerCase(unsigned long pString) {
	unsigned long i=0, cnt=0;
	while(((char*)pString)[i]) {
		if((((char*)pString)[i] >= 0x41) && (((char*)pString)[i] <= 0x5a)) {	/* between A..Z */
			((char*)pString)[i] += 0x20;
			cnt++;
		}
		i++;
	}
	return cnt;
}
```

#### brdkStrToUpperCase.c
```c
#include <brdkSTR_func.h>

signed long brdkStrToUpperCase(unsigned long pString) {
	unsigned long i=0,cnt=0;
	while(((char*)pString)[i]) {
		if((((char*)pString)[i] >= 0x61) && (((char*)pString)[i] <= 0x7a)) {	/* between a..z */
			((char*)pString)[i] -= 0x20;
			cnt++;
		}
		i++;
	}
	return cnt;
}
```

#### brdkStrToUpperCaseWords.c
```c
#include <brdkSTR_func.h>

signed long brdkStrToUpperCaseWords(unsigned long pString) {
	unsigned long i=0,cnt=0;
	if(((char*)pString)[i]) {
		if(((char*)pString)[i] >= 0x61 && ((char*)pString)[i] <= 0x7a) {	/* check the first character */
	 		((char*)pString)[i] -= 0x20;
			cnt++;
		}
	}
	i++;
	while(((char*)pString)[i]) {
		if((((char*)pString)[i] >= 0x61) && (((char*)pString)[i] <= 0x7a) && ((char*)pString)[i-1] == 0x20){	/* between a..z and a space before */
			((char*)pString)[i] -= 0x20;
			cnt++;
		}
		i++;
	}
	return cnt;
}
```

#### brdkStrTrim.c
```c
#include <brdkSTR_func.h>

signed long brdkStrTrim(unsigned long pString, signed long direction) {
	signed long i,j=0,len;
	if(direction == BRDK_STR_BOTH_TRIM || direction == BRDK_STR_LEFT_TRIM) {
		len = brdkStrLen(pString);
		while(((char*)pString)[0] == 0x20) {									/* white space */
			for(i=0;i < len;i++) ((char*)pString)[i] = ((char*)pString)[i+1];	/* moves all characters one place left */
			len--;
			j++;
		}
	}
	if(direction == BRDK_STR_BOTH_TRIM || direction == BRDK_STR_RIGHT_TRIM) {
		len = brdkStrLen(pString)-1;
		while(((char*)pString)[len] == 0x20 && len > -1) {						/* white space */
			((char*)pString)[len--] = 0;
			j++;
		}
	}
	return j;
}
```

#### brdkStrUdintToA.c
```c
#include <brdkSTR_func.h>

signed long brdkStrUdintToA(unsigned long value, unsigned long pString, unsigned char base) {
	int i=0;
	((char*)pString)[0] = 0;
	base = !base ? 10 : base;	/* make sure base is not 0 */
	if (value != 0) {
		while (value > 0) {
			unsigned long rem = value % base;
	       	((char*)pString)[i++] = (rem > 9)? (rem-10) + 0x41 : rem + 0x30;	/* 0x41 = A, 0x30 = 0*/
	       	value = value/base;
		}
		((char*)pString)[i] = 0;
	}
	else {
		((char*)pString)[i++] = 0x30;	/* 0 */
		((char*)pString)[i] = 0;
	}
	brdkStrReverse(pString,0,-1);
	return i;
}
```

#### brdkStrWord.c
```c
#include <brdkSTR_func.h>

signed long brdkStrWord(unsigned long pDestination, unsigned long pSource, unsigned long pDelimiter, signed long number, unsigned long sizeOfString) {
	unsigned long sIdx = 0, dIdx = 0;
	signed long cnt = 1;
	if(pDestination != 0 && pSource != 0 && number != 0) {
		if(pDelimiter == 0) pDelimiter = (unsigned long)" ";			/* use white space is delimiter pointer is 0 */
		while(((char*)pSource)[sIdx] != 0) {
			if(((char*)pSource)[sIdx] != ((char*)pDelimiter)[0]) {
				((char*)pDestination)[dIdx++] = ((char*)pSource)[sIdx];
			}
			else {
				if(number > 0) {
					if(cnt == number) break;
					else {
						dIdx = 0;
						cnt++;
					}
				}
				else {
					cnt = number;
					dIdx = 0;
				}
			}
			sIdx++;
			if(dIdx > sizeOfString) return -2;								/* destination string too small */
		}
		if(number > cnt) return -3;
		((char*)pDestination)[dIdx] = 0;
		return dIdx;
	}
	else return -1;
	return -4;
}
```

#### brdkSTR_func.h
```c
#ifndef BRDK_STR_FUNCS
#define BRDK_STR_FUNCS 1

#include <brdkSTR.h>
#include <bur/plctypes.h>

#ifdef __cplusplus
	extern "C"
	{
#endif

signed long search(signed long pString, signed long lenString, signed long pSearchString, signed long lenSearch);
unsigned long aToUdint(unsigned long pString, signed long len, unsigned char base);

#ifdef __cplusplus
	};
#endif

#endif
```

#### brdkSTR_func.c
```c
#include <brdkSTR_func.h>

/* search for a string in a string */
signed long search(signed long pString, signed long lenString, signed long pSearchString, signed long lenSearch) {
	signed long pos=-1, i=0,j=0;
	if(lenString>lenSearch) {
		for(i=0; i <= lenString-lenSearch; i++) {
			j=0;
			if(((char*)pString)[i] == ((char*)pSearchString)[j]) {
				while(((char*)pString)[i+j] == ((char*)pSearchString)[j]) {
					j++;
					if(j==lenSearch) {
						pos = i;
						i=lenString-lenSearch+1;
						break;
					}
				}
			}
		}
	}
	return pos;
}

/* convert a string to an UDINT */
unsigned long aToUdint(unsigned long pString, signed long len, unsigned char base) {
	unsigned long value = 0,i;
	if(len > 0) {
		for(i=0; i <len; i++) {
			switch(base) {

				case 0: case 10:
					if(((char*)pString)[i] >= 0x30 && ((char*)pString)[i] <= 0x39) value = (value * 10) + (((char*)pString)[i]-0x30);			/* 0x30 = 0, 0x39 = 9 */
					else {
						value = 0;
						i = len;
					}
					break;

				case 2:
					if(((char*)pString)[i] >= 0x30 && ((char*)pString)[i] <= 0x31) value += (((char*)pString)[i]-0x30)*(1<<(len-1-i));			/* 0x30 = 0, 0x31 = 1 */
					else {
						value = 0;
						i = len;
					}
					break;

				case 16:
					if(((char*)pString)[i] >= 0x30 && ((char*)pString)[i] <= 0x39) 	value += (((char*)pString)[i]-0x30)*(1<<(4*(len-1-i)));		/* 0x30 = 0, 0x39 = 9 */
					else if(((char*)pString)[i] >= 0x41 && ((char*)pString)[i] <= 0x46) value += (((char*)pString)[i]-0x37)*(1<<(4*(len-1-i)));	/* 0x41 = A, 0x46 = F */
					else if(((char*)pString)[i] >= 0x61 && ((char*)pString)[i] <= 0x66)value += (((char*)pString)[i]-0x57)*(1<<(4*(len-1-i)));	/* 0x61 = a, 0x66 = f */
					else {
						value = 0;
						i = len;
					}
					break;

				default:
					value = 0;
					i = len;
					break;

			}
		}
	}
	return value;
}
```

- CHANGELOG - brdkSTR change log (not shown)

- LICENSE - brdkSTR license (not shown)

### Library Logical/Libraries/brdk/brdkUSB (ANSIC, version 1.00.2)
Depends on: AsUSB, FileIO

#### brdkUSB.typ - Exported data types
```iecst
TYPE
	brdk_usb_status_typ :
		( (*Status of the function block*)
		BRDK_USB_STATUS_NO_USB_DEV_FOUND, (*No USB device found*)
		BRDK_USB_STATUS_FB_READY (*Ready to connect*)
		);
	brdk_usb_connect_node_output_typ : 	STRUCT  (*Node device info*)
		device : STRING[5]; (*Node device name*)
		freeMemory : DINT; (*[Mb] -1 means memory info could not be read*)
		totalMemory : DINT; (*[Mb] -1 means memory info could not be read*)
	END_STRUCT;
	brdk_usb_connect_internal_typ : 	STRUCT  (*internal variables*)
		UsbNodeListGet_0 : UsbNodeListGet; (*get node list*)
		nodeIdBuffer : ARRAY[0..BRDK_USB_MAX_DEVICES]OF UDINT; (*node id buffer*)
		oldCnt : UDINT; (*old count*)
		node : ARRAY[0..BRDK_USB_MAX_DEVICES]OF brdk_usb_connect_int_node_typ; (*node list*)
		simulationMountActivated : BOOL; (*is the mount being simulated*)
	END_STRUCT;
	brdk_usb_connect_int_node_typ : 	STRUCT  (*internal node variables*)
		state : UINT; (*node state*)
		infoBuffer : usbNode_typ; (*node info*)
		UsbNodeGet_0 : UsbNodeGet; (*usb get node*)
		DevLink_0 : DevLink; (*creates a deveice link*)
		DevUnlink_0 : DevUnlink; (*unlinks a device link*)
		DevMemInfo_0 : DevMemInfo; (*reads the memory info about the device*)
		device : STRING[8]; (*device name*)
		param : STRING[20]; (*device parameters*)
		devLinkFailCnt : UDINT; (*faild dev link count*)
	END_STRUCT;
END_TYPE
```

#### brdkUSB.var - Exported constants
```iecst
VAR CONSTANT
	BRDK_USB_MAX_DEVICES : UINT := 4; (*Maximum numbers of connected USB devices. 4 means 5*)
END_VAR
```

#### brdkUSB.fun - Exported functions and function blocks
```iecst
FUNCTION_BLOCK brdkUSBConnect (*This function block outputs a list of all connected USB flash devices with a connected device name that can be used in e.g. FileIO library. B&R technology guards are filtered away from the node list.*)
	VAR_INPUT
		updateMemInfo : BOOL; (*Updates the memory info of the nodes*)
		simulateMount : BOOL; (*Simulates a USB mount. Creates a file device for C:\USB\*)
	END_VAR
	VAR_OUTPUT
		node : ARRAY[0..BRDK_USB_MAX_DEVICES] OF brdk_usb_connect_node_output_typ; (*List of avaible USB nodes*)
		status : brdk_usb_status_typ; (*Status of the function block*)
	END_VAR
	VAR
		internal : brdk_usb_connect_internal_typ; (*internal variables*)
	END_VAR
END_FUNCTION_BLOCK
```

#### brdkUSBConnect.c
```c
#include <bur/plctypes.h>
#include <string.h>
#ifdef __cplusplus
	extern "C"
	{
#endif

	#include "brdkUSB.h"

#ifdef __cplusplus
	};
#endif

#define true 1
#define false 0

/* Converts an UDINT into a STRING type */
static unsigned char brdkUSBuditoa(unsigned long Value, char* pString) {
	int i, j=0;
	pString[0] = 0;
	if (Value > 0) {
		while (Value > 0) {
			j++;
			for(i=j; i > 0 ; i--) {
				pString[i] =pString[i-1];
			}
			pString[0] = (Value % 10) + 48;			/* ASCII 48-57 = 0..9 */
			Value = (Value / 10);
		}
	}
	else {
		pString[0] = 48;								/* adds just a zero char  */
		pString[1] = 0;								/* ends the string  */
		j = 1;
	}
	return j;
}

void brdkUSBConnect(struct brdkUSBConnect* inst) {
	brdk_usb_connect_internal_typ* this = &inst->internal;
	int i;
	char tmp[2];

	/* get list of all connected usb nodes */
	this->UsbNodeListGet_0.enable 					= true;
	this->UsbNodeListGet_0.pBuffer					= (UDINT)&this->nodeIdBuffer;
	this->UsbNodeListGet_0.bufferSize 				= sizeof(this->nodeIdBuffer);
	this->UsbNodeListGet_0.filterInterfaceClass 	= asusb_CLASS_MASS_STORAGE;
	this->UsbNodeListGet_0.filterInterfaceSubClass 	= 0;
	UsbNodeListGet(&this->UsbNodeListGet_0);
	if(this->UsbNodeListGet_0.status == ERR_OK) {
		if(this->oldCnt != this->UsbNodeListGet_0.listNodes && this->UsbNodeListGet_0.listNodes > 0) {
			/* find an avaible node index */
			if(this->oldCnt < this->UsbNodeListGet_0.listNodes) {
				for(i=0; i<= BRDK_USB_MAX_DEVICES; i++) {
					if(this->node[i].UsbNodeGet_0.nodeId == 0) {
						this->node[i].UsbNodeGet_0.nodeId = this->nodeIdBuffer[this->UsbNodeListGet_0.listNodes-1];
						break;
					}
				}
			}
		}
	}
	else if(inst->simulateMount && !this->simulationMountActivated) {
	/* find an avaible node index */
		for(i=0; i<= BRDK_USB_MAX_DEVICES; i++) {
			if(this->node[i].UsbNodeGet_0.nodeId == 0) {
				this->node[i].UsbNodeGet_0.nodeId = 4294967295LL;
				this->simulationMountActivated = true;
				break;
			}
		}
	}
	this->oldCnt = this->UsbNodeListGet_0.listNodes;

	/* state machine for all usb nodes */
	for(i=0; i<= BRDK_USB_MAX_DEVICES; i++) {

		switch(this->node[i].state) {

			case 0: /* wait for id */
				if(this->node[i].UsbNodeGet_0.nodeId != 0) {
					this->node[i].UsbNodeGet_0.enable 		= (this->node[i].UsbNodeGet_0.nodeId < 4294967294LL);
					this->node[i].UsbNodeGet_0.pBuffer 		= (UDINT)&this->node[i].infoBuffer;
					this->node[i].UsbNodeGet_0.bufferSize 	= sizeof(usbNode_typ);
					UsbNodeGet(&this->node[i].UsbNodeGet_0);
					this->node[i].state 					= 10;
				}
				break;

			case 10:	/* get usb node info (interface name) */
				UsbNodeGet(&this->node[i].UsbNodeGet_0);
				switch(this->node[i].UsbNodeGet_0.status) {

					case ERR_OK:
						/* filter B&R technology guard from list */
						if(this->node[i].infoBuffer.vendorId == 1615 && this->node[i].infoBuffer.productId == 1001) this->node[i].state = 70;
						else {
							strcpy(this->node[i].device,"USB");
							brdkUSBuditoa(i,tmp);
							strcat(this->node[i].device,tmp);
							this->node[i].DevLink_0.pDevice = (UDINT)&this->node[i].device;
							strcpy(this->node[i].param, "/DEVICE=");
							strcat(this->node[i].param, this->node[i].infoBuffer.ifName);
							this->node[i].DevLink_0.pParam = (UDINT)&this->node[i].param;
							this->node[i].DevLink_0.enable = true;
							this->node[i].state = 20;
						}
						break;

					case asusbERR_USB_NOTFOUND:
						this->node[i].UsbNodeGet_0.nodeId = 0;
						memset(&this->node[i].infoBuffer,0,sizeof(usbNode_typ));
						this->node[i].state = 0;
						break;

					case ERR_FUB_ENABLE_FALSE:
						strcpy(this->node[i].device,"USB");
						brdkUSBuditoa(i,tmp);
						strcat(this->node[i].device,tmp);
						this->node[i].DevLink_0.pDevice = (UDINT)&this->node[i].device;
						strcpy(this->node[i].param, "/DEVICE=C:\\USB");
						this->node[i].DevLink_0.pParam = (UDINT)&this->node[i].param;
						this->node[i].DevLink_0.enable = true;
						this->node[i].state = 20;
						break;

				}
				break;

			case 20:	/* create device link */
				DevLink(&this->node[i].DevLink_0);
				switch(this->node[i].DevLink_0.status) {

					case ERR_OK:
						strcpy(inst->node[i].device,this->node[i].device);
						this->node[i].state = 40;
						break;

					case fiERR_DEVICE_ALREADY_EXIST:
						this->node[i].DevUnlink_0.enable 	= 1;
						this->node[i].DevUnlink_0.handle 	= this->node[i].DevLink_0.handle;
						this->node[i].state 				= 30;
						break;
				}
				break;

			case 30:	/* unlink device link */
				DevUnlink(&this->node[i].DevUnlink_0);
				switch(this->node[i].DevUnlink_0.status ) {

					case ERR_OK: case fiERR_DEVICE_INVALID_HANDLE:
						this->node[i].DevUnlink_0.enable 	= 0;
						DevUnlink(&this->node[i].DevUnlink_0);
						this->node[i].DevLink_0.enable 		= 0;
						DevLink(&this->node[i].DevLink_0);
						this->node[i].DevLink_0.enable 		= 1;
						this->node[i].devLinkFailCnt++;
						brdkUSBuditoa(this->node[i].devLinkFailCnt,tmp);
						strcat(this->node[i].device,tmp);
						this->node[i].DevLink_0.pDevice 	= (UDINT)&this->node[i].device;
						this->node[i].state					= 20;
						break;

				}
				break;

			case 40:	/* usb node ready - monitor node */
				UsbNodeGet(&this->node[i].UsbNodeGet_0);
				switch(this->node[i].UsbNodeGet_0.status) {

					case ERR_OK:
						if(inst->updateMemInfo || inst->node[i].totalMemory == 0) {
							this->node[i].DevMemInfo_0.enable = true;
							this->node[i].DevMemInfo_0.pDevice = this->node[i].DevLink_0.pDevice;
							this->node[i].state = 50;
						}
						break;

					case asusbERR_USB_NOTFOUND:
						strcpy(inst->node[i].device,"");
						this->node[i].DevUnlink_0.enable 	= true;
						this->node[i].DevUnlink_0.handle 	= this->node[i].DevLink_0.handle;
						this->node[i].state = 60;
						break;

					case ERR_FUB_ENABLE_FALSE:
						if(!inst->simulateMount && this->simulationMountActivated) {
							strcpy(inst->node[i].device,"");
							this->node[i].DevUnlink_0.enable 	= true;
							this->node[i].DevUnlink_0.handle 	= this->node[i].DevLink_0.handle;
							this->simulationMountActivated 		= false;
							this->node[i].state = 60;
						}
						break;

				}
				break;

			case 50:	/* read meminfo */
				DevMemInfo(&this->node[i].DevMemInfo_0);
				switch(this->node[i].DevMemInfo_0.status) {

					case ERR_OK:
						inst->node[i].freeMemory 	= this->node[i].DevMemInfo_0.freemem/1048576;	/* output must be in mb */
						inst->node[i].totalMemory 	= this->node[i].DevMemInfo_0.memsize/1048576;	/* output must be in mb */
						this->node[i].state 		= 40;
						break;

					case fiERR_DETMEMINFO: case fiERR_DEVICE_MANAGER:
						inst->node[i].freeMemory 	= -1;	/* output must be in mb */
						inst->node[i].totalMemory 	= -1;	/* output must be in mb */
						this->node[i].state 		= 40;
						break;

					case ERR_FUB_BUSY: break;
					default: this->node[i].state = 40; break;
				}
				break;

			case 60:	/* unlink device */
				DevUnlink(&this->node[i].DevUnlink_0);
				switch(this->node[i].DevUnlink_0.status ) {

					case ERR_OK: case fiERR_DEVICE_INVALID_HANDLE:
						this->node[i].DevUnlink_0.enable 	= false;
						DevUnlink(&this->node[i].DevUnlink_0);
						this->node[i].DevLink_0.enable 		= false;
						DevLink(&this->node[i].DevLink_0);
						this->node[i].UsbNodeGet_0.nodeId = 0;
						memset(&this->node[i].infoBuffer,0,sizeof(usbNode_typ));
						inst->node[i].freeMemory 	= 0;
						inst->node[i].totalMemory 	= 0;
						this->node[i].state = 0;
						break;

				}
				break;

			case 70:	/* B&R technology guard state */
				UsbNodeGet(&this->node[i].UsbNodeGet_0);
				switch(this->node[i].UsbNodeGet_0.status) {

					case ERR_OK: break;

					case asusbERR_USB_NOTFOUND:
						this->node[i].UsbNodeGet_0.nodeId = 0;
						memset(&this->node[i].infoBuffer,0,sizeof(usbNode_typ));
						this->node[i].state = 0;
						break;

				}
				break;

			case 1000:	/* simulate usb device */

				break;

		}
	}

	/* output status */
	for(i=0; i<= BRDK_USB_MAX_DEVICES; i++) {
		if(inst->node[i].device[0] != 0) {
			inst->status = BRDK_USB_STATUS_FB_READY;
			break;
		}
		else inst->status = BRDK_USB_STATUS_NO_USB_DEV_FOUND;
	}

	inst->updateMemInfo = 0;	/* reset update command */

}
```

- LICENSE (not shown)

- CHANGELOG - brdkUSB change log (not shown)

### Library Logical/Libraries/brdk/brdkFile (ANSIC, version 0.00.2)
Depends on: AsIODiag, AsUSB, FileIO, brdkSTR

#### brdkFile.typ - Data types
```iecst
TYPE
	brdk_file_dev_handler_int_typ : 	STRUCT  (*Internal variables.*)
		fileState : UINT; (*State of the file device handler.*)
		driveState : UINT; (*State of the drive handler.*)
		DevLink_0 : DevLink; (*Device link.*)
		DevUnlink_0 : DevUnlink; (*Device unlink.*)
		DirInfo_0 : DirInfo; (*Directory create.*)
		drive : STRING[30]; (*Drive.*)
		deviceParam : STRING[BRDK_FILE_MAX_PATH_LEN]; (*Device parameter string.*)
		fileIdx : DINT; (*File index.*)
		activeHandles : ARRAY[0..BRDK_FILE_MAX_FILES_DEVICES]OF UDINT; (*Active handles.*)
		driveReady : BOOL; (*Drive ready to use.*)
		oldUseUSB : BOOL; (*Holds the old command.*)
		usbOK : BOOL; (*USB drive present and ready to use.*)
		brdkFileCreateSubFolders_0 : brdkFileCreateSubFolders; (*Create sub folders.*)
		UsbNodeListGet_0 : UsbNodeListGet; (*Get list of USB nodes.*)
		UsbNodeGet_0 : UsbNodeGet; (*Get USB node.*)
		nodeId : ARRAY[0..BRDK_FILE_MAX_USB_NODES]OF UDINT; (*Node id buffer list.*)
		nodeIdx : USINT; (*Node id index.*)
		usbNode : usbNode_typ; (*Node info.*)
		oldUSBok : BOOL; (*Holds the old status.*)
		oldNodeId : UDINT; (*Holds the old node id.*)
	END_STRUCT;
	brdk_file_dev_handler_sim_typ : 	STRUCT  (*Simulation options.*)
		pcRootFolder : STRING[BRDK_FILE_MAX_PATH_LEN] := 'plcRoot'; (*Path on the PC that will simulate the root of the controller. Default plcRoot -> C:\plcRoot\*)
		pcUSBDrive : brdk_file_drive_typ := D_DRIVE; (*Drive letter of the PC's USB. Default D:\.*)
		pcHDDrive : brdk_file_drive_typ := C_DRIVE; (*Drive letter of the PC's HD. Default C:\.*)
	END_STRUCT;
	brdk_file_dev_handler_setup_typ : 	STRUCT  (*Setup options.*)
		plcDrive : brdk_file_drive_typ := C_DRIVE; (*Drive letter of the controller flash. Default C:\.*)
		usbOverrule : BOOL := FALSE; (*Inserted USB stick will overrule internal flash if the USB stick is present.*)
		fileDevices : ARRAY[0..BRDK_FILE_MAX_FILES_DEVICES]OF brdk_file_file_devices_typ := [(name:='CONFIG',path:='config'),(name:='RECIPES',path:='recipes'),8((0))]; (*File devices. Default CONFIG and RECEIPES with config and recipes folder.*)
		rootFileDeviceName : STRING[10] := 'ROOT';
	END_STRUCT;
	brdk_file_drive_typ :
		( (*Drive selection. Default C:\.*)
		C_DRIVE := 0, (*C:\*)
		D_DRIVE := 1, (*D:\*)
		E_DRIVE := 2, (*E:\*)
		F_DRIVE := 3, (*F:\*)
		G_DRIVE := 4 (*G:\*)
		) := C_DRIVE;
	brdk_file_file_devices_typ : 	STRUCT  (*File devices setup.*)
		name : STRING[BRFK_FILE_MAX_FILE_DEVICE_LEN]; (*Name of the file device to be used as input for file functions.*)
		path : STRING[BRDK_FILE_MAX_PATH_LEN]; (*Folder path for the file device. Only the folders must be entered the drive is setup in the setup options. E.g. config.*)
	END_STRUCT;
	brdk_file_create_subfold_int_typ : 	STRUCT  (*Internal variables.*)
		state : DINT; (*State of the function block.*)
		DirCreate_0 : DirCreate; (*Directory create.*)
		tmpPath : STRING[BRDK_FILE_MAX_PATH_LEN]; (*Temp path string.*)
		pathPos : DINT; (*Path position.*)
		tmpPathPos : DINT; (*Tmp path position.*)
		tmpLen : DINT; (*Temp length.*)
	END_STRUCT;
	brdk_file_read_internal_typ : 	STRUCT  (*Internal variables.*)
		state : DINT; (*State of the function block.*)
		FileOpen_0 : FileOpen; (*File open.*)
		FileClose_0 : FileClose; (*File close.*)
		FileReadEx_0 : FileReadEx; (*File read.*)
		offset : UDINT; (*Read offset.*)
	END_STRUCT;
	brdk_file_write_internal_typ : 	STRUCT  (*Internal variables.*)
		state : DINT; (*State of the function block.*)
		FileOpen_0 : FileOpen; (*File open.*)
		FileCreate_0 : FileCreate; (*File create.*)
		FileClose_0 : FileClose; (*File close.*)
		FileDelete_0 : FileDelete; (*File delete.*)
		FileWrite_0 : FileWrite; (*File write.*)
	END_STRUCT;
END_TYPE
```

#### brdkFile.var - Constants
```iecst
VAR CONSTANT
	BRDK_FILE_MAX_USB_NODES : USINT := 5; (*Maximum number of connected USB nodes. (5 means 6)*)
	BRDK_FILE_MAX_FILES_DEVICES : USINT := 15; (*Maximum numbers of file devices. (9 means 10)*)
	BRDK_FILE_MAX_PATH_LEN : UINT := 200; (*Maximum length of a path.*)
	BRFK_FILE_MAX_FILE_DEVICE_LEN : UINT := 50; (*Maximum length of file device names.*)
END_VAR
```

#### brdkFile.fun - Functions and function blocks
```iecst
FUNCTION_BLOCK brdkFileDeviceHandler (*Easy file device handler. This function block makes file device handling easy. The idea of the function block is that you only need to create one file device name that can be used for both internal and usb flash.*) (*$GROUP=User,$CAT=User,$GROUPICON=User.png,$CATICON=User.png*)
	VAR_INPUT
		enable : BOOL; (*Enables the function block.*)
		setup : brdk_file_dev_handler_setup_typ; (*Setup options.*)
		simulation : brdk_file_dev_handler_sim_typ; (*Simulation options.*)
		useUSB : BOOL; (*Stores on the USB if it is possible. Can be auto selected in the setup options.*)
	END_VAR
	VAR_OUTPUT
		availableDevices : ARRAY[0..BRDK_FILE_MAX_FILES_DEVICES] OF STRING[BRFK_FILE_MAX_FILE_DEVICE_LEN]; (*List of available file devices.*)
		ready : BOOL; (*Means that all file devices have been created and are ready to use.*)
		description : STRING[200]; (*Status description.*)
		status : UINT; (*Status of FileIO function blocks.*)
	END_VAR
	VAR
		internal : brdk_file_dev_handler_int_typ; (*Internal variables.*)
	END_VAR
END_FUNCTION_BLOCK

FUNCTION_BLOCK brdkFileCreateSubFolders (*Creates folders based on a path string.*) (*$GROUP=User,$CAT=User,$GROUPICON=User.png,$CATICON=User.png*)
	VAR_INPUT
		enable : BOOL; (*Enables the function block.*)
		path : STRING[BRDK_FILE_MAX_PATH_LEN]; (*Path of folder to be created. Use \ to seperate folders.*)
		fileDevice : STRING[BRFK_FILE_MAX_FILE_DEVICE_LEN]; (*File device name.*)
	END_VAR
	VAR_OUTPUT
		description : STRING[200]; (*Status description.*)
		done : BOOL; (*Function block done.*)
		status : UINT; (*Status of DirCreate function block.*)
	END_VAR
	VAR
		internal : brdk_file_create_subfold_int_typ; (*Internal variables.*)
	END_VAR
END_FUNCTION_BLOCK

FUNCTION_BLOCK brdkFileWrite (*Write data to a file.*) (*$GROUP=User,$CAT=User,$GROUPICON=User.png,$CATICON=User.png*)
	VAR_INPUT
		enable : BOOL; (*Enables the function block.*)
		fileDevice : STRING[BRFK_FILE_MAX_FILE_DEVICE_LEN]; (*File device name.*)
		fileName : STRING[BRDK_FILE_MAX_PATH_LEN]; (*File name. If the file does not exist it will be created.*)
		pData : UDINT; (*Pointer to the data that must be written to the file.*)
		dataLength : UDINT; (*Length of the data that must be written. If 0 is specified \0 will end the data.*)
		overwrite : BOOL; (*Overwrite existing file. If not set the data will be appended to existing file.*)
	END_VAR
	VAR_OUTPUT
		description : STRING[200]; (*Status description.*)
		done : BOOL; (*Function block done.*)
		status : UINT; (*Status of FileIO function blocks.*)
	END_VAR
	VAR
		internal : brdk_file_write_internal_typ; (*Internal variables.*)
	END_VAR
END_FUNCTION_BLOCK

FUNCTION_BLOCK brdkFileRead (*Read data from a file.*) (*$GROUP=User,$CAT=User,$GROUPICON=User.png,$CATICON=User.png*)
	VAR_INPUT
		enable : BOOL; (*Enables the function block.*)
		fileDevice : STRING[BRFK_FILE_MAX_FILE_DEVICE_LEN]; (*File device name.*)
		fileName : STRING[BRDK_FILE_MAX_PATH_LEN]; (*File name. If the file does not exist it will be created.*)
		pData : UDINT; (*Pointer to the data where the data is read to.*)
		dataLength : UDINT; (*Length of the read data buffer.*)
	END_VAR
	VAR_OUTPUT
		description : STRING[200]; (*Status description.*)
		bytesread : UDINT;
		done : BOOL; (*Function block done.*)
		status : UINT; (*Status of FileIO function blocks.*)
	END_VAR
	VAR
		internal : brdk_file_read_internal_typ; (*Internal variables.*)
	END_VAR
END_FUNCTION_BLOCK
```

#### brdkFileDeviceHandler.c - Easy file device handler.
```c
#include <brdkFile_func.h>

#define BR_TG_VENDOR_ID 1615
#define BR_TG_PRODUCT_ID 1001

void brdkFileDeviceHandler(struct brdkFileDeviceHandler* inst) {
	brdk_file_dev_handler_int_typ* this = (brdk_file_dev_handler_int_typ*)&inst->internal;		/* pointer to the internal structure */
	brdk_file_dev_handler_setup_typ* setup = (brdk_file_dev_handler_setup_typ*)&inst->setup;	/* pointer to the setup structure */
	brdk_file_dev_handler_sim_typ* sim = (brdk_file_dev_handler_sim_typ*)&inst->simulation;		/* pointer to the simulation structure */
	char tmpStr[200];

	if(inst->enable) {

		/* check weither the controller is beeing simulated and watch the usb status */
		if(!DiagCpuIsSimulated()) {
			if(!this->UsbNodeGet_0.enable) this->UsbNodeListGet_0.enable = true;
			this->UsbNodeListGet_0.pBuffer					= (unsigned long)&this->nodeId;
			this->UsbNodeListGet_0.bufferSize 				= sizeof(this->nodeId);
			this->UsbNodeListGet_0.filterInterfaceClass 	= asusb_CLASS_MASS_STORAGE;
			this->UsbNodeListGet_0.filterInterfaceSubClass 	= asusb_SUBCLASS_SCSI_COMMAND_SET;
			UsbNodeListGet(&this->UsbNodeListGet_0);
			if(this->UsbNodeListGet_0.status == asusbERR_USB_NOTFOUND) {
				this->nodeIdx = 0;
				this->usbOK = false;
			}

			this->UsbNodeGet_0.enable 		= true;
			this->UsbNodeGet_0.nodeId 		= this->nodeId[this->nodeIdx];
			this->UsbNodeGet_0.pBuffer 		= (unsigned long)&this->usbNode;
			this->UsbNodeGet_0.bufferSize 	= sizeof(this->usbNode);
			UsbNodeGet(&this->UsbNodeGet_0);
			if(this->UsbNodeGet_0.status == ERR_OK) {
				if(this->usbNode.vendorId == BR_TG_VENDOR_ID && this->usbNode.productId == BR_TG_PRODUCT_ID) {
					this->UsbNodeGet_0.enable 		= false;
					UsbNodeGet(&this->UsbNodeGet_0);
					this->nodeIdx++;
				}
				else this->usbOK = true;
			}
			else if(this->UsbNodeGet_0.status == asusbERR_USB_NOTFOUND) {
				this->UsbNodeListGet_0.enable = true;
				this->nodeIdx = 0;
				this->usbOK = false;
			}
			if(this->oldNodeId != this->UsbNodeGet_0.nodeId) this->usbOK = false;
			this->oldNodeId = this->UsbNodeGet_0.nodeId;
		}
		else {
			/* look for USB root folder */
			if(this->DirInfo_0.pDevice != 0) {
				this->DirInfo_0.enable 	= true;
				this->DirInfo_0.pPath 	= (unsigned long)"";
				DirInfo(&this->DirInfo_0);
				switch(this->DirInfo_0.status) {
					case 0: this->usbOK = true; break;
					case 20723: this->usbOK = false; break;
					default: break;
				}
			}
		}
		if(setup->usbOverrule) inst->useUSB = this->usbOK;	/* USB stick will overrule */
	}
	else {
		this->usbOK 					= false;
		this->nodeIdx 					= 0;
		this->DirInfo_0.enable 			= false;
		DirInfo(&this->DirInfo_0);
		this->UsbNodeGet_0.enable 		= false;
		UsbNodeGet(&this->UsbNodeGet_0);
		this->UsbNodeListGet_0.enable 	= false;
		UsbNodeListGet(&this->UsbNodeListGet_0);
	}

	/* drive handler */
	switch(this->driveState) {

		case 0:
			if(inst->enable) {
				if(!DiagCpuIsSimulated()) {	/* check if the controller is simulated */
					if((inst->useUSB && this->usbOK) || !inst->useUSB) {
						this->driveReady = true;
						if(!inst->useUSB) getDrive(setup->plcDrive,this->drive);
						else brdkStrCpy((unsigned long)this->drive,(unsigned long)this->usbNode.ifName);
						this->driveState = 499;
					}
				}
				else {
					this->DevLink_0.enable 	= true;
					this->DevLink_0.pDevice = (unsigned long)"INTUSB";
					this->DevLink_0.pParam 	= buildParameterString(getDrive(sim->pcUSBDrive,this->drive),(char*)&"",(char*)&this->deviceParam);
					this->driveState 		= 100;
				}
			}
			break;

		case 100:	/* create a file device for finding an attached usb flash */
			DevLink(&this->DevLink_0);
			if(this->DevLink_0.status != ERR_FUB_BUSY) {
				if(this->DevLink_0.status == ERR_OK || this->DevLink_0.status == fiERR_DEVICE_ALREADY_EXIST) {
					this->DirInfo_0.pDevice = this->DevLink_0.pDevice;
					this->DevLink_0.enable 	= false;
					DevLink(&this->DevLink_0);
					this->driveState 		= 110;
				}
				else {
					inst->status = this->DevLink_0.status;
					this->DevLink_0.enable 	= false;
					DevLink(&this->DevLink_0);
					brdkStrCpy((unsigned long)inst->description,(unsigned long)"error calling DevLink. Flip enable to reset fb.");
					this->driveState = 900;
				}
			}
			break;

		case 110:	/* wait for DirInfo to have been call once. Fb is call above */
			switch(this->DirInfo_0.status) {

				case 0: case 20723:
					if(!inst->useUSB) {
						getDrive(sim->pcHDDrive,this->drive);
						brdkStrCat((unsigned long)this->drive,(unsigned long)sim->pcRootFolder);
					}
					else getDrive(sim->pcUSBDrive,this->drive);
					this->driveState = 499;
					this->driveReady = true;
					break;

				case 65534: case 65535: break;

				default:
					inst->status 			= this->DirInfo_0.status;
					this->DirInfo_0.enable 	= false;
					DirInfo(&this->DirInfo_0);
					brdkStrCpy((unsigned long)inst->description,(unsigned long)"error calling DirInfo. Flip enable to reset fb.");
					this->driveReady = false;
					this->driveState = 900;
					break;

			}
			break;

		case 499:	/* waiting for file devices to be ready */
			if(!inst->enable) {
				this->driveReady = false;
				this->driveState = 900;
			}
			else if(inst->ready) this->driveState = 500;
			break;

		case 500:	/* check if USB status changes */
			if(!inst->enable) {
				this->driveReady = false;
				this->driveState = 900;
			}
			else if((this->oldUseUSB != inst->useUSB) || (inst->useUSB && (this->oldUSBok != this->usbOK))) {	/* usb must be used and the ok status has changed */
				this->driveReady = false;
				if(inst->useUSB && !this->usbOK) brdkStrCpy((unsigned long)inst->description,(unsigned long)"USB not ready. Turn off useUSB command.");
				else this->driveState = 510;
			}
			this->oldUseUSB = inst->useUSB;
			this->oldUSBok 	= this->usbOK;
			this->oldNodeId = this->UsbNodeGet_0.nodeId;
			break;

		case 510:	/* select the new drive */
			if(!DiagCpuIsSimulated()) {	/* check if the controller is simulated */
				if(!inst->useUSB) getDrive(setup->plcDrive,this->drive);
				else brdkStrCpy((unsigned long)this->drive,(unsigned long)this->usbNode.ifName);
			}
			else {
				if(!inst->useUSB) {
					getDrive(sim->pcHDDrive,this->drive);
					brdkStrCat((unsigned long)this->drive,(unsigned long)sim->pcRootFolder);
				}
				else getDrive(sim->pcUSBDrive,this->drive);
			}
			this->driveReady = true;
			this->driveState = 499;
			break;

		case 900:	/* error state */
			this->driveReady = false;
			if(!inst->enable) {
				inst->status 		= 0;
				this->driveState 	= 0;
			}
			break;

	}

	/* file device handler */
	switch(this->fileState) {

		case 0:	/* wait for a drive */
			if(inst->enable) {
				if(this->driveReady) {
					this->DevLink_0.enable 	= true;

					this->DevLink_0.pDevice = (unsigned long)&inst->setup.rootFileDeviceName;
					this->DevLink_0.pParam 	= buildParameterString((char*)&this->drive,(char*)&"",(char*)&this->deviceParam);
					this->fileState 		= 10;
				}
			}
			else {
				inst->ready = false;
			}
			break;

		case 10:
			brdkStrCpy((unsigned long)inst->description,(unsigned long)"creates a devlink for the drive root");
			DevLink(&this->DevLink_0);
			if(this->DevLink_0.status != ERR_FUB_BUSY) {
				if(this->DevLink_0.status == ERR_OK) {

					brdkStrCpy((unsigned long)inst->availableDevices[0],this->DevLink_0.pDevice);
					this->activeHandles[0] = this->DevLink_0.handle;
					this->DevLink_0.enable 	= false;
					DevLink(&this->DevLink_0);
					this->fileIdx = 0;
					if(setup->fileDevices[this->fileIdx].name[0] != 0 && setup->fileDevices[this->fileIdx].path[0] != 0) {
						brdkStrCpy((unsigned long)this->brdkFileCreateSubFolders_0.path,(unsigned long)setup->fileDevices[this->fileIdx].path);
						brdkStrCpy((unsigned long)this->brdkFileCreateSubFolders_0.fileDevice,this->DevLink_0.pDevice);
						this->brdkFileCreateSubFolders_0.enable = true;
						brdkFileCreateSubFolders(&this->brdkFileCreateSubFolders_0);
						this->fileState = 20;
					}
					else this->fileState = 100;
				}
				else if(this->DevLink_0.status == fiERR_DEVICE_ALREADY_EXIST) {
					if(this->DevLink_0.handle != 0) {
						inst->status = this->DevLink_0.status;
						this->DevLink_0.enable 	= false;
						DevLink(&this->DevLink_0);
						brdkStrCpy((unsigned long)inst->description,(unsigned long)"Device ");
						brdkStrCat((unsigned long)inst->description,this->DevLink_0.pDevice);
						brdkStrCat((unsigned long)inst->description,(unsigned long)" already exists. Reboot controller to kill the old device.");
						this->fileState = 900;
					}
					else {
						this->DevUnlink_0.enable = true;
						this->DevUnlink_0.handle = this->DevLink_0.handle;
						this->DevLink_0.enable 	= false;
						DevLink(&this->DevLink_0);
						this->fileState = 40;
					}
				}
				else {
					brdkStrCpy((unsigned long)inst->description,(unsigned long)"error calling DevLink. Flip enable to reset fb.");
					inst->status 			= this->DevLink_0.status;
					this->DevLink_0.enable 	= false;
					DevLink(&this->DevLink_0);
					this->fileState 		= 900;
				}
			}
			break;

		case 20:
			brdkStrCpy((unsigned long)inst->description,(unsigned long)"creates the needed folders");
			brdkFileCreateSubFolders(&this->brdkFileCreateSubFolders_0);
			if(this->brdkFileCreateSubFolders_0.done) {
				this->brdkFileCreateSubFolders_0.enable = false;
				brdkFileCreateSubFolders(&this->brdkFileCreateSubFolders_0);
				this->fileIdx++;
				if(setup->fileDevices[this->fileIdx].name[0] != 0 && setup->fileDevices[this->fileIdx].path[0] != 0) {
					this->brdkFileCreateSubFolders_0.enable = true;
					brdkStrCpy((unsigned long)this->brdkFileCreateSubFolders_0.path,(unsigned long)setup->fileDevices[this->fileIdx].path);
					brdkFileCreateSubFolders(&this->brdkFileCreateSubFolders_0);
				}
				else {
					this->fileIdx = 0;
					this->DevLink_0.enable 	= true;
					this->DevLink_0.pDevice = (unsigned long)setup->fileDevices[this->fileIdx].name;
					this->DevLink_0.pParam 	= buildParameterString((char*)&this->drive,(char*)&setup->fileDevices[this->fileIdx].path,(char*)&this->deviceParam);
					this->fileState = 30;
				}
			}
			else if(this->brdkFileCreateSubFolders_0.status == fiERR_FILE_DEVICE) {
				if(DiagCpuIsSimulated()) {
					this->DevUnlink_0.enable 	= true;
					this->DevUnlink_0.handle 	= this->activeHandles[0];
					this->activeHandles[0] 		= 0;
					DevUnlink(&this->DevUnlink_0);
					this->brdkFileCreateSubFolders_0.enable = false;
					brdkFileCreateSubFolders(&this->brdkFileCreateSubFolders_0);
					this->fileState 			= 200;
				}
				else {
					brdkStrCpy((unsigned long)inst->description,(unsigned long)"error calling brdkFileCreateSubFolders. Flip enable to reset fb.");
					inst->status 				= this->brdkFileCreateSubFolders_0.status;
					this->brdkFileCreateSubFolders_0.enable = false;
					brdkFileCreateSubFolders(&this->brdkFileCreateSubFolders_0);
					this->fileState 			= 900;
				}
			}
			else if(this->brdkFileCreateSubFolders_0.status != ERR_FUB_BUSY) brdkStrCpy((unsigned long)inst->description,(unsigned long)"error calling brdkFileCreateSubFolders. Check fb for error codes.");
			break;

		case 30:
			brdkStrCpy((unsigned long)inst->description,(unsigned long)"creates the needed file devices");
			DevLink(&this->DevLink_0);
			if(this->DevLink_0.status != ERR_FUB_BUSY) {
				if(this->DevLink_0.status == ERR_OK) {
					brdkStrCpy((unsigned long)inst->availableDevices[this->fileIdx+1],this->DevLink_0.pDevice);
					this->activeHandles[this->fileIdx+1] = this->DevLink_0.handle;
					this->DevLink_0.enable 	= false;
					DevLink(&this->DevLink_0);
					this->fileIdx++;
					if(setup->fileDevices[this->fileIdx].name[0] != 0 && setup->fileDevices[this->fileIdx].path[0] != 0) {
						this->DevLink_0.enable 	= true;
						this->DevLink_0.pDevice = (unsigned long)setup->fileDevices[this->fileIdx].name;
						this->DevLink_0.pParam 	= buildParameterString((char*)&this->drive,(char*)&setup->fileDevices[this->fileIdx].path,(char*)&this->deviceParam);
					}
					else {
						inst->ready = true;
						brdkStrCpy((unsigned long)inst->description,(unsigned long)"all file devices are ready to use");
						this->fileState = 100;
					}
				}
				else {
					brdkStrCpy((unsigned long)inst->description,(unsigned long)"error calling DevLink. Flip enable to reset fb.");
					inst->status 			= this->DevLink_0.status;
					this->DevLink_0.enable 	= false;
					DevLink(&this->DevLink_0);
					this->fileState 		= 900;
				}
			}
			break;

		case 40:
			DevUnlink(&this->DevUnlink_0);
			if(this->DevUnlink_0.status != ERR_FUB_BUSY) {
				if(this->DevUnlink_0.status == ERR_OK) {
					this->DevUnlink_0.enable = false;
					DevUnlink(&this->DevUnlink_0);
					this->DevLink_0.enable 	= true;
					this->DevLink_0.pDevice = (unsigned long)&inst->setup.rootFileDeviceName;
					this->DevLink_0.pParam 	= buildParameterString((char*)&this->drive,(char*)&"",(char*)&this->deviceParam);
					this->fileState 		= 10;
				}
				else {
					brdkStrCpy((unsigned long)inst->description,(unsigned long)"error calling DevUnlink. Flip enable to reset fb.");
					inst->status 				= this->DevUnlink_0.status;
					this->DevUnlink_0.enable 	= false;
					DevUnlink(&this->DevUnlink_0);
					this->fileState 			= 900;
				}
			}
			break;

		case 100:	/* wait for interuption */
			if(!inst->enable) {
				inst->ready 	= false;
				this->fileState = 900;
			}
			if(!this->driveReady) {
				inst->ready = false;
				if(this->activeHandles[0] != 0) {
					this->fileIdx = 0;
					this->DevUnlink_0.enable 	= true;
					this->DevUnlink_0.handle 	= this->activeHandles[this->fileIdx];
					this->fileState 			= 110;
				}
				else this->fileState = 0;
			}
			break;

		case 110:	/* unlink file devices */
			DevUnlink(&this->DevUnlink_0);
			if(this->DevUnlink_0.status != ERR_FUB_BUSY) {
				if(this->DevUnlink_0.status == ERR_OK) {
					brdkStrCpy((unsigned long)inst->availableDevices[this->fileIdx],(unsigned long)"");
					this->activeHandles[this->fileIdx] = 0;
					this->fileIdx++;
					this->DevUnlink_0.enable = false;
					DevUnlink(&this->DevUnlink_0);
					if(this->activeHandles[this->fileIdx] != 0) {
						this->DevUnlink_0.enable = true;
						this->DevUnlink_0.handle = this->activeHandles[this->fileIdx];
					}
					else this->fileState = 0;
				}
				else {
					brdkStrCpy((unsigned long)inst->description,(unsigned long)"error calling DevUnlink. Flip enable to reset fb.");
					inst->status 				= this->DevUnlink_0.status;
					this->DevUnlink_0.enable 	= false;
					DevUnlink(&this->DevUnlink_0);
					this->fileState 			= 900;
				}
			}
			break;

		case 200:
			DevUnlink(&this->DevUnlink_0);
			if(this->DevUnlink_0.status != ERR_FUB_BUSY) {
				if(this->DevUnlink_0.status == ERR_OK) {
					this->DevUnlink_0.enable = false;
					DevUnlink(&this->DevUnlink_0);
					this->DevLink_0.enable 	= true;
					this->DevLink_0.pDevice = (unsigned long)"tmpRoot";
					this->DevLink_0.pParam 	= buildParameterString(getDrive(sim->pcHDDrive,tmpStr),(char*)&"",(char*)&this->deviceParam);
					this->fileState 		= 210;
				}
				else {
					brdkStrCpy((unsigned long)inst->description,(unsigned long)"error calling DevUnlink. Flip enable to reset fb.");
					inst->status 				= this->DevUnlink_0.status;
					this->DevUnlink_0.enable 	= false;
					DevUnlink(&this->DevUnlink_0);
					this->fileState 			= 900;
				}
			}
			break;

		case 210:
			brdkStrCpy((unsigned long)inst->description,(unsigned long)"creates a file devive for sim root folder");
			DevLink(&this->DevLink_0);
			if(this->DevLink_0.status != ERR_FUB_BUSY) {
				if(this->DevLink_0.status == ERR_OK) {
					this->DevUnlink_0.handle 	= this->DevLink_0.handle;
					this->DevLink_0.enable 		= false;
					DevLink(&this->DevLink_0);
					this->brdkFileCreateSubFolders_0.enable = true;
					brdkStrCpy((unsigned long)this->brdkFileCreateSubFolders_0.path,(unsigned long)sim->pcRootFolder);
					brdkStrCpy((unsigned long)this->brdkFileCreateSubFolders_0.fileDevice,this->DevLink_0.pDevice);
					brdkFileCreateSubFolders(&this->brdkFileCreateSubFolders_0);
					this->fileState 			= 220;
				}
				else {
					brdkStrCpy((unsigned long)inst->description,(unsigned long)"error calling DevLink. Flip enable to reset fb.");
					inst->status 				= this->DevLink_0.status;
					this->DevLink_0.enable 		= false;
					DevLink(&this->DevLink_0);
					this->fileState 			= 900;
				}
			}
			break;

		case 220:
			brdkStrCpy((unsigned long)inst->description,(unsigned long)"creates the needed folders");
			brdkFileCreateSubFolders(&this->brdkFileCreateSubFolders_0);
			if(this->brdkFileCreateSubFolders_0.done) {
				this->brdkFileCreateSubFolders_0.enable = false;
				brdkFileCreateSubFolders(&this->brdkFileCreateSubFolders_0);
				this->DevUnlink_0.enable 	= true;
				this->fileState				= 230;
			}
			else if(this->brdkFileCreateSubFolders_0.status != ERR_FUB_BUSY) {
				brdkStrCpy((unsigned long)inst->description,(unsigned long)"error calling brdkFileCreateSubFolders. Flip enable to reset fb.");
				inst->status 				= this->brdkFileCreateSubFolders_0.status;
				this->brdkFileCreateSubFolders_0.enable = false;
				brdkFileCreateSubFolders(&this->brdkFileCreateSubFolders_0);
				this->fileState 			= 900;
			}
			break;

		case 230:
			DevUnlink(&this->DevUnlink_0);
			if(this->DevUnlink_0.status != ERR_FUB_BUSY) {
				if(this->DevUnlink_0.status == ERR_OK) {
					this->DevUnlink_0.enable = false;
					DevUnlink(&this->DevUnlink_0);
					this->fileState 			= 0;
				}
				else {
					inst->status 				= this->DevUnlink_0.status;
					this->DevUnlink_0.enable 	= false;
					DevUnlink(&this->DevUnlink_0);
					brdkStrCpy((unsigned long)inst->description,(unsigned long)"error calling DevUnlink. Flip enable to reset fb.");
					this->fileState 			= 900;
				}
			}
			break;

		case 900: /* error state */
			if(!inst->enable) {
				inst->status 	= 0;
				this->fileState = 0;
			}
			break;

	}

}
```

#### brdkFileCreateSubFolders.c - Creates folders based on a path string.
```c
#include <brdkFile_func.h>

void brdkFileCreateSubFolders(struct brdkFileCreateSubFolders* inst) {
	brdk_file_create_subfold_int_typ* this = (brdk_file_create_subfold_int_typ*)&inst->internal;

	switch(this->state) {

		case 0:
			if(inst->enable) {
				this->DirCreate_0.pDevice 	= (unsigned long)inst->fileDevice;
				this->DirCreate_0.pName 	= (unsigned long)this->tmpPath;
				brdkStrMemSet((unsigned long)&this->tmpPath,0,sizeof(this->tmpPath));
				brdkStrReplace((unsigned long)inst->path,(unsigned long)"/",(unsigned long)"\\");	/* replace all / with \ */
				this->pathPos = 0;
				if(inst->path[0] == 0x5c) this->pathPos = 1;
				this->tmpPathPos = 0;
				while(inst->path[this->pathPos] != 0) {
					this->DirCreate_0.enable 			= true;
					if(inst->path[this->pathPos] == 0x5c) {
						this->tmpPath[this->tmpPathPos++] 	= inst->path[this->pathPos++];
						break;
					}
					else this->tmpPath[this->tmpPathPos++] = inst->path[this->pathPos++];
				}
				if(this->DirCreate_0.enable) {
					DirCreate(&this->DirCreate_0);
					this->state = 10;
				}
				else {
					inst->done = true;
					this->state = 100;
				}
			}
			break;

		case 10:
			brdkStrCpy((unsigned long)inst->description,(unsigned long)"creates the needed folders");
			DirCreate(&this->DirCreate_0);
			if(this->DirCreate_0.status != ERR_FUB_BUSY) {
				if(this->DirCreate_0.status == ERR_OK || this->DirCreate_0.status == fiERR_DIR_ALREADY_EXIST) {
					this->DirCreate_0.enable 	= false;
					DirCreate(&this->DirCreate_0);
					while(inst->path[this->pathPos] != 0) {
						this->DirCreate_0.enable 			= true;
						if(inst->path[this->pathPos] == 0x5c) {
							this->tmpPath[this->tmpPathPos++] 	= inst->path[this->pathPos++];
							break;
						}
						else {
							this->tmpPath[this->tmpPathPos++] 	= inst->path[this->pathPos++];
							this->DirCreate_0.enable 			= true;
						}
					}
					if(this->DirCreate_0.enable) DirCreate(&this->DirCreate_0);
					else {
						inst->done = true;
						this->state = 100;
					}
				}
				else {
					brdkStrCpy((unsigned long)inst->description,(unsigned long)"error calling DirCreate. Check fb for error codes.");
					inst->status = this->DirCreate_0.status;
					this->state = 100;
				}
			}
			break;

		case 100:
			if(inst->status == ERR_OK) brdkStrCpy((unsigned long)inst->description,(unsigned long)"done. Flip and set enable to restart");
			if(!inst->enable) {
				inst->done 				= false;
				inst->status 			= 0;
				inst->description[0] 	= 0;
				this->state 			= 0;
			}
			break;

	}
}
```

#### brdkFileWrite.c - Write data to a file.
```c
#include <brdkFile_func.h>

void brdkFileWrite(struct brdkFileWrite* inst) {
	brdk_file_write_internal_typ* this = (brdk_file_write_internal_typ*)&inst->internal;

	switch(this->state) {

		case 0:
			brdkStrCpy((unsigned long)inst->description,(unsigned long)"waiting for FB to be enabled.");
			if(inst->enable) {
				brdkStrCpy((unsigned long)inst->description,(unsigned long)"fb busy.");
				this->FileCreate_0.enable 	= true;
				this->FileCreate_0.pDevice 	= (unsigned long)&inst->fileDevice;
				this->FileCreate_0.pFile 	= (unsigned long)&inst->fileName;
				FileCreate(&this->FileCreate_0);
				this->state 				= 10;
			}
			inst->done					= false;
			break;

		case 10:
			brdkStrCpy((unsigned long)inst->description,(unsigned long)"waiting for FileCreate to be done.");
			FileCreate(&this->FileCreate_0);
			switch(this->FileCreate_0.status) {

				case 0:	/* ERR_OK */
					this->FileWrite_0.enable 	= true;
					this->FileWrite_0.ident 	= this->FileCreate_0.ident;
					this->FileWrite_0.offset 	= 0;
					this->FileWrite_0.pSrc 		= inst->pData;
					this->FileWrite_0.len 		= inst->dataLength != 0 ? inst->dataLength : brdkStrLen(inst->pData);
					this->FileCreate_0.enable 	= false;
					FileCreate(&this->FileCreate_0);
					FileWrite(&this->FileWrite_0);
					this->state 				= 40;
					break;

				case 20705: /* fiERR_EXIST  */
					if(!inst->overwrite) {
						this->FileOpen_0.enable 	= true;
						this->FileOpen_0.pDevice 	= (unsigned long)&inst->fileDevice;
						this->FileOpen_0.pFile 		= (unsigned long)&inst->fileName;
						this->FileOpen_0.mode 		= fiWRITE_ONLY;
						FileOpen(&this->FileOpen_0);
						this->state 				= 20;
					}
					else {
						this->FileDelete_0.enable 	= true;
						this->FileDelete_0.pDevice 	= (unsigned long)&inst->fileDevice;
						this->FileDelete_0.pName 	= (unsigned long)&inst->fileName;
						FileDelete(&this->FileDelete_0);
						this->state = 30;
					}
					break;

				case 65535: break;	/* ERR_FUB_BUSY */

				default:
					brdkStrCpy((unsigned long)inst->description,(unsigned long)"error FileCreate. check status. Flip enable to reset fb.");
					inst->status 				= this->FileCreate_0.status;
					this->FileCreate_0.enable 	= false;
					FileCreate(&this->FileCreate_0);
					this->state 				= 60;
					break;

			}
			break;

		case 20:
			brdkStrCpy((unsigned long)inst->description,(unsigned long)"waiting for FileOpen to be done.");
			FileOpen(&this->FileOpen_0);
			switch(this->FileOpen_0.status) {

				case 0:	/* ERR_OK */
					this->FileWrite_0.enable 	= true;
					this->FileWrite_0.ident 	= this->FileOpen_0.ident;
					this->FileWrite_0.offset 	= this->FileOpen_0.filelen;
					this->FileWrite_0.pSrc 		= inst->pData;
					this->FileWrite_0.len 		= inst->dataLength != 0 ? inst->dataLength : brdkStrLen(inst->pData);
					this->FileOpen_0.enable = false;
					FileOpen(&this->FileOpen_0);
					FileWrite(&this->FileWrite_0);
					this->state 				= 40;
					break;

				case 65535: break;	/* ERR_FUB_BUSY */

				default:
					brdkStrCpy((unsigned long)inst->description,(unsigned long)"error FileOpen. check status. Flip enable to reset fb.");
					inst->status 				= this->FileOpen_0.status;
					this->FileOpen_0.enable = false;
					FileOpen(&this->FileOpen_0);
					this->state 				= 60;
					break;

			}
			break;

		case 30:
			brdkStrCpy((unsigned long)inst->description,(unsigned long)"waiting for FileDelete to be done.");
			FileDelete(&this->FileDelete_0);
			switch(this->FileDelete_0.status) {

				case 0:	case 20708: /* ERR_OK - fiERR_FILE_NOT_FOUND */
					this->FileDelete_0.enable = false;
					FileDelete(&this->FileDelete_0);
					this->FileCreate_0.enable 	= true;
					this->FileCreate_0.pDevice 	= (unsigned long)&inst->fileDevice;
					this->FileCreate_0.pFile 	= (unsigned long)&inst->fileName;
					FileCreate(&this->FileCreate_0);
					this->state 				= 10;
					break;

				case 65535: break;	/* ERR_FUB_BUSY */

				default:
					brdkStrCpy((unsigned long)inst->description,(unsigned long)"error FileDelete. check status. Flip enable to reset fb.");
					inst->status 				= this->FileDelete_0.status;
					this->FileDelete_0.enable = false;
					FileDelete(&this->FileDelete_0);
					this->state 				= 60;
					break;

			}
			break;

		case 40:
			brdkStrCpy((unsigned long)inst->description,(unsigned long)"waiting for FileWrite to be done.");
			FileWrite(&this->FileWrite_0);
			switch(this->FileWrite_0.status) {

				case 0:	/* ERR_OK */
					this->FileWrite_0.enable 	= false;
					FileWrite(&this->FileWrite_0);
					this->FileClose_0.enable 	= true;
					this->FileClose_0.ident 	= this->FileWrite_0.ident;
					FileClose(&this->FileClose_0);
					this->state 				= 50;
					break;

				case 65535: break;	/* ERR_FUB_BUSY */

				default:
					brdkStrCpy((unsigned long)inst->description,(unsigned long)"error FileWrite. check status. Flip enable to reset fb.");
					inst->status 				= this->FileWrite_0.status;
					this->FileWrite_0.enable 	= false;
					FileWrite(&this->FileWrite_0);
					this->state 				= 60;
					break;

			}
			break;

		case 50:
			brdkStrCpy((unsigned long)inst->description,(unsigned long)"waiting for FileClose to be done.");
			FileClose(&this->FileClose_0);
			switch(this->FileClose_0.status) {

				case 0:	case 20721: /* ERR_OK - fiERR_FILE_NOT_OPENED */
					this->FileClose_0.enable 	= false;
					FileClose(&this->FileClose_0);
					inst->done					= true;
					brdkStrCpy((unsigned long)inst->description,(unsigned long)"fb done. Flip enable and set to start fb again.");
					this->state 				= 60;
					break;

				case 65535: break;	/* ERR_FUB_BUSY */

				default:
					brdkStrCpy((unsigned long)inst->description,(unsigned long)"error FileClose. check status. Flip enable to reset fb.");
					inst->status 				= this->FileClose_0.status;
					this->FileClose_0.enable 	= false;
					FileClose(&this->FileClose_0);
					this->state 				= 60;
					break;

			}
			break;

		case 60:
			if(!inst->enable) {
				inst->done		= false;
				inst->status	= 0;
				this->state 	= 0;
			}
			break;

	}

}
```

#### brdkFileRead.c - Read data from a file.
```c
#include <brdkFile_func.h>

void brdkFileRead(struct brdkFileRead* inst) {
	brdk_file_read_internal_typ* this = (brdk_file_read_internal_typ*)&inst->internal;

	switch(this->state) {

		case 0:
			brdkStrCpy((unsigned long)inst->description,(unsigned long)"waiting for FB to be enabled.");
			if(inst->enable) {
				inst->bytesread = 0;
				if(inst->dataLength > 0) {
					brdkStrCpy((unsigned long)inst->description,(unsigned long)"fb busy.");
					this->FileOpen_0.enable 	= true;
					this->FileOpen_0.pDevice 	= (unsigned long)&inst->fileDevice;
					this->FileOpen_0.pFile 		= (unsigned long)&inst->fileName;
					this->FileOpen_0.mode 		= fiREAD_ONLY;
					FileOpen(&this->FileOpen_0);
					this->state 				= 10;
				}
				else {
					brdkStrCpy((unsigned long)inst->description,(unsigned long)"datalength = 0. Set dataLength to buffer size. Flip enable to reset fb.");
					this->state 				= 40;
				}
			}
			inst->done					= false;
			break;

		case 10:
			brdkStrCpy((unsigned long)inst->description,(unsigned long)"waiting for FileOpen to be done.");
			FileOpen(&this->FileOpen_0);
			switch(this->FileOpen_0.status) {

				case 0:	/* ERR_OK */
					this->FileReadEx_0.enable 	= true;
					this->FileReadEx_0.ident 		= this->FileOpen_0.ident;
					this->FileReadEx_0.offset 	= 0;
					this->FileReadEx_0.pDest 		= inst->pData;
					this->FileReadEx_0.len 		= inst->dataLength;
					this->FileOpen_0.enable 	= false;
					FileOpen(&this->FileOpen_0);
					FileReadEx(&this->FileReadEx_0);
					this->state 				= 20;
					break;

				case 65535: break;	/* ERR_FUB_BUSY */

				default:
					brdkStrCpy((unsigned long)inst->description,(unsigned long)"error FileOpen. check status. Flip enable to reset fb.");
					inst->status 				= this->FileOpen_0.status;
					this->FileOpen_0.enable 	= false;
					FileOpen(&this->FileOpen_0);
					this->state 				= 40;
					break;

			}
			break;

		case 20:
			brdkStrCpy((unsigned long)inst->description,(unsigned long)"waiting for FileRead to be done.");
			FileReadEx(&this->FileReadEx_0);
			switch(this->FileReadEx_0.status) {

				case 0:	/* ERR_OK */
					inst->bytesread = this->FileReadEx_0.bytesread;
					this->FileReadEx_0.enable 	= false;
					FileReadEx(&this->FileReadEx_0);
					this->FileClose_0.enable 	= true;
					this->FileClose_0.ident 	= this->FileReadEx_0.ident;
					FileClose(&this->FileClose_0);
					this->state 				= 30;
					break;

				case 65535: break;	/* ERR_FUB_BUSY */

				default:
					brdkStrCpy((unsigned long)inst->description,(unsigned long)"error FileClose. check status. Flip enable to reset fb.");
					inst->status 				= this->FileReadEx_0.status;
					this->FileReadEx_0.enable 	= false;
					FileRead(&this->FileReadEx_0);
					this->state 				= 40;
					break;

			}
			break;

		case 30:
			brdkStrCpy((unsigned long)inst->description,(unsigned long)"waiting for FileClose to be done.");
			FileClose(&this->FileClose_0);
			switch(this->FileClose_0.status) {

				case 0:	case 20721: /* ERR_OK - fiERR_FILE_NOT_OPENED */
					this->FileClose_0.enable 	= false;
					FileClose(&this->FileClose_0);
					inst->done					= true;
					brdkStrCpy((unsigned long)inst->description,(unsigned long)"fb done. Flip enable and set to start fb again.");
					this->state 				= 40;
					break;

				case 65535: break;	/* ERR_FUB_BUSY */

				default:
					brdkStrCpy((unsigned long)inst->description,(unsigned long)"error FileClose. check status. Flip enable to reset fb.");
					inst->status 				= this->FileClose_0.status;
					this->FileClose_0.enable 	= false;
					FileClose(&this->FileClose_0);
					this->state 				= 40;
					break;

			}
			break;

		case 40:
			if(!inst->enable) {
				inst->done					= false;
				inst->status				= 0;
				this->state 				= 0;
			}
			break;

	}

}
```
